// TIA Portal project "Proyecto1" (V15)

(* hardware
DEVICE "S7-1200 station_1"  S7-1200 Station
   slot 0: "Rack_0"  S7-1200 Rack  Rack  V1.0
   slot 1: "PLC_1"  CPU 1214C AC/DC/Rly  6ES7 214-1BG40-0XB0  V4.2
   slot 3: "CB 1241 (RS485)"  CB 1241 (RS485)  6ES7 241-1CH30-1XB0  V1.0
DEVICE "HMI_1"  KTP600 Basic color PN
   slot 0: "HMI_1"  KTP600 Basic color PN  6AV6 647-0AD11-3AX0  12.0.0.0
   slot 1: "HMI_RT_1"  KTP600 Basic color PN  6AV6 647-0AD11-3AX0  12.0.0.0
   slot 5: "HMI_1.IE_CP_1"  PROFINET Interface  12.0.0.0
      slot 1: "Interfaz PROFINET_1"  PROFINET Interface
         slot 1: "Port_1"  Port
*)

// ===== PLC "PLC_1"  CPU 1214C AC/DC/Rly =====

VAR_GLOBAL   // PLC tag table "Tabla de variables estándar"
   "First Scan" AT %M1.0 : Bool;
   "Tag_1" AT %I0.1 : Bool;
   "Tag_2" AT %I0.2 : Bool;
   "Tag_3" AT %Q0.0 : Bool;
   "0.5 Hz clock" AT %M0.7 : Bool;
   "mHora" AT %M0.3 : Bool;
   "reset_hora_contador" AT %MW100 : Int;
END_VAR

TYPE "FLOW_PARA_DB"
   STRUCT
      "Process Values" : Struct
         Massflow : Real;
         Volumeflow : Real;
         Density : Real;
         Temperature : Real;
         "Frame temperature" : Real;
      END_STRUCT;
      "Identification data" : Struct
         "Sensor serial number" : String[20];
      END_STRUCT;
      Totalizer : Struct
         "Totalizer value" : Real;
         "Reset totalizer" : UInt := 1;
      END_STRUCT;
      "Device diagnostic" : Struct
         "Driver current" : Real;
         "Pick-up amplitude 1" : Real;
         "Pick-up amplitude 2" : Real;
         "Sensor frequency" : Real;
      END_STRUCT;
      "Zero Point adjustment" : Struct
         "Zero point duration" : UInt := 30;
         "Standard deviation" : Real;
         "Zero point offset value" : Real;
         "Zero point adjust progress" : UInt;
         "Zero point adjust status" : UInt;
         "Start Zero point adjustment" : UInt := 2;
      END_STRUCT;
      Setup : Struct
         "Flow direction" : UInt := 0;
         "Process noise damping" : UInt;
         "Low Massflow cutofff" : Real;
         "Low volumeflow cutoff" : Real;
      END_STRUCT;
      "Aerated Flow" : Struct
         "Aerated flow alarm limit" : UInt;
         "Aerated flow warning limit" : UInt;
         "Measurement sample time" : UInt;
         "Aerated flow filter" : UInt;
         "Filter time constant" : UInt;
         "Filter start hysteresis" : Real;
         "Minimum filtering time" : UInt;
      END_STRUCT;
      Alarms : Struct
         "Alarm group 1" : UDInt;
         "Alarm group 2" : UDInt;
      END_STRUCT;
      "Access level" : Struct
         "Access level" : UInt;
         "Access Password" : UInt := 2457;
      END_STRUCT;
      HMI_Commands : Struct
         CMD_200 : Bool;
         CMD_210 : Bool;
         CMD_220 : Bool;
         CMD_230 : Bool;
         CMD_240 : Bool;
         CMD_250 : Bool;
         CMD_260 : Bool;
         CMD_280 : Bool;
         CMD_290 : Bool;
         CMD_420 : Bool;
         CMD_440 : Bool;
         CMD_450 : Bool;
         CMD_460 : Bool;
         CMD_490_log_in : Bool;
         CMD_491_log_out : Bool;
      END_STRUCT;
      FB_Interface : Struct
         Input : Struct
            MB_ADDR : UInt := 3;
            CMD_IN : Int;
         END_STRUCT;
         Output : Struct
            CMD_INPR : Bool;
            CMD_ERR : Bool;
            ERR_MB_MASTER : Bool;
            STATUS_MB_MASTER : Word;
         END_STRUCT;
         InOut : Struct
            CMD_EN : Bool;
         END_STRUCT;
      END_STRUCT;
   END_STRUCT;
END_TYPE

DATA_BLOCK "FECHA_Y_HORA"   // DB2
{ S7_Optimized_Access := 'TRUE' }
VERSION : 0.1
   VAR
      Local : DTL;
   END_VAR
BEGIN
END_DATA_BLOCK

DATA_BLOCK "CONTADOR_DB"   // DB3
{ S7_Optimized_Access := 'TRUE' }
VERSION : 0.1
// stored: InstanceOfName CONTADOR
"CONTADOR"
BEGIN
END_DATA_BLOCK

DATA_BLOCK "CONTADOR_NODE"   // DB5
{ S7_Optimized_Access := 'FALSE' }
VERSION : 0.1
   VAR
      cSecadero : Int;
      cHorno : Int;
   END_VAR
BEGIN
END_DATA_BLOCK

DATA_BLOCK "DB_FLOW_PARA"   // DB17
{ S7_Optimized_Access := 'FALSE' }
VERSION : 0.1
BEGIN
END_DATA_BLOCK

DATA_BLOCK "FC410_FC_MODBUS_DB"   // DB95
{ S7_Optimized_Access := 'TRUE' }
VERSION : 0.1
// stored: InstanceOfName FC410_MODBUS
"FC410_MODBUS"
BEGIN
END_DATA_BLOCK

// folder: System blocks/Program resources

DATA_BLOCK "CONTADOR_PIEZAS_SECADERO"   // DB1
{ S7_Optimized_Access := 'TRUE' }
AUTHOR : Simatic
FAMILY : IEC
NAME : CNTR
VERSION : 1.0
// stored: InstanceOfName IEC_COUNTER
"IEC_COUNTER"
BEGIN
END_DATA_BLOCK

DATA_BLOCK "CONTADOR_PIEZAS_HORNO"   // DB4
{ S7_Optimized_Access := 'TRUE' }
AUTHOR : Simatic
FAMILY : IEC
NAME : CNTR
VERSION : 1.0
// stored: InstanceOfName IEC_COUNTER
"IEC_COUNTER"
BEGIN
END_DATA_BLOCK

// folder: (top level)

FUNCTION_BLOCK "FC410_MODBUS"   // FB1, LAD
{ S7_Optimized_Access := 'TRUE' }
VERSION : 0.1
   VAR_INPUT
      CMD_IN : Int;
      MB_ADDR : UInt;
   END_VAR
   VAR_OUTPUT
      CMD_INPR : Bool;
      CMD_ERR : Bool;
      ERR_MB_MASTER : Bool;
      STATUS_MB_MASTER : Word;
   END_VAR
   VAR_IN_OUT
      CMD_EN : Bool;
      DB_PARA : "FLOW_PARA_DB";
   END_VAR
   VAR
      CMD_INPR_COUNT : USInt;
   END_VAR
   VAR_TEMP
      Temp_Length_Read : DInt;
      "Temp_String Help" : String[2];
      "Alarm Group 2_temp" : UDInt;
   END_VAR
   VAR_TEMP   // added for the SCL form of the ladder/FBD networks
      _w1 : Bool;
      _w2 : Bool;
   END_VAR
BEGIN

REGION Network 1: Command 200 - Read Process Values 1/3
   // Reading Massflow, Volumeflow and density
   // 
   // DATA_ADDR: Modbus adr.: 3000 + 3002 + 3004
   // DATA_LEN: 6 words
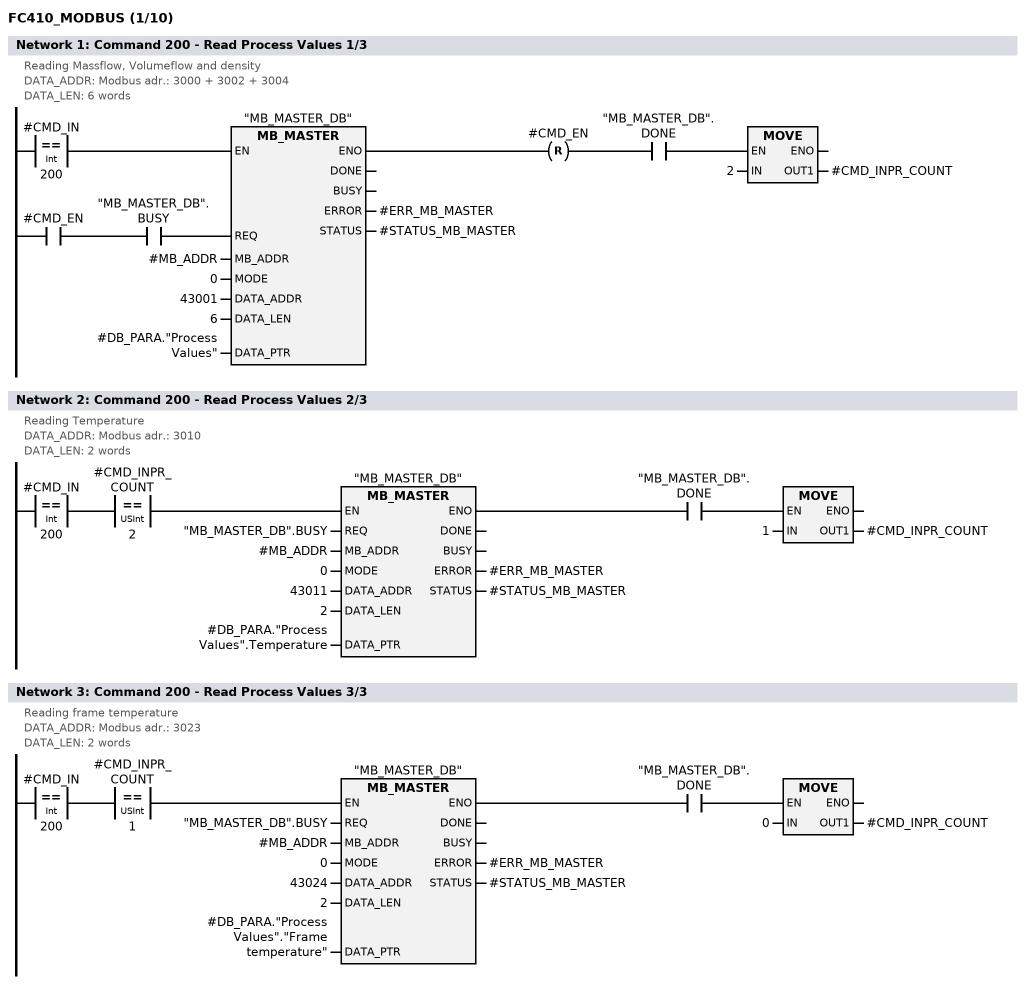
   // ENO of a box is taken as its EN; it also drops when the box reports an error
   #_w1 := #CMD_IN = 200;
   IF #_w1 THEN
       "MB_MASTER_DB"(REQ := #CMD_EN AND "MB_MASTER_DB".BUSY,   // MB_MASTER
                      MB_ADDR := #MB_ADDR,
                      MODE := 0,
                      DATA_ADDR := 43001,
                      DATA_LEN := 6,
                      DATA_PTR := #DB_PARA."Process Values",
                      ERROR => #ERR_MB_MASTER,
                      STATUS => #STATUS_MB_MASTER);
       #CMD_EN := FALSE;
   END_IF;
   IF #_w1 AND "MB_MASTER_DB".DONE THEN #CMD_INPR_COUNT := 2; END_IF;
END_REGION

REGION Network 2: Command 200 - Read Process Values 2/3
   // Reading Temperature
   // 
   // DATA_ADDR: Modbus adr.: 3010
   // DATA_LEN: 2 words
   // ENO of a box is taken as its EN; it also drops when the box reports an error
   #_w1 := (#CMD_IN = 200) AND (#CMD_INPR_COUNT = 2);
   IF #_w1 THEN
       "MB_MASTER_DB"(REQ := "MB_MASTER_DB".BUSY,   // MB_MASTER
                      MB_ADDR := #MB_ADDR,
                      MODE := 0,
                      DATA_ADDR := 43011,
                      DATA_LEN := 2,
                      DATA_PTR := #DB_PARA."Process Values".Temperature,
                      ERROR => #ERR_MB_MASTER,
                      STATUS => #STATUS_MB_MASTER);
   END_IF;
   IF #_w1 AND "MB_MASTER_DB".DONE THEN #CMD_INPR_COUNT := 1; END_IF;
END_REGION

REGION Network 3: Command 200 - Read Process Values 3/3
   // Reading frame temperature
   // 
   // DATA_ADDR: Modbus adr.: 3023
   // DATA_LEN: 2 words
   // ENO of a box is taken as its EN; it also drops when the box reports an error
   #_w1 := (#CMD_IN = 200) AND (#CMD_INPR_COUNT = 1);
   IF #_w1 THEN
       "MB_MASTER_DB"(REQ := "MB_MASTER_DB".BUSY,   // MB_MASTER
                      MB_ADDR := #MB_ADDR,
                      MODE := 0,
                      DATA_ADDR := 43024,
                      DATA_LEN := 2,
                      DATA_PTR := #DB_PARA."Process Values"."Frame temperature",
                      ERROR => #ERR_MB_MASTER,
                      STATUS => #STATUS_MB_MASTER);
   END_IF;
   IF #_w1 AND "MB_MASTER_DB".DONE THEN #CMD_INPR_COUNT := 0; END_IF;
END_REGION

REGION Network 4: Command 210 - Read Sensor Serial Number
   // DATA_ADDR: Modbus adr.: 4033
   // DATA_LEN: 10 words
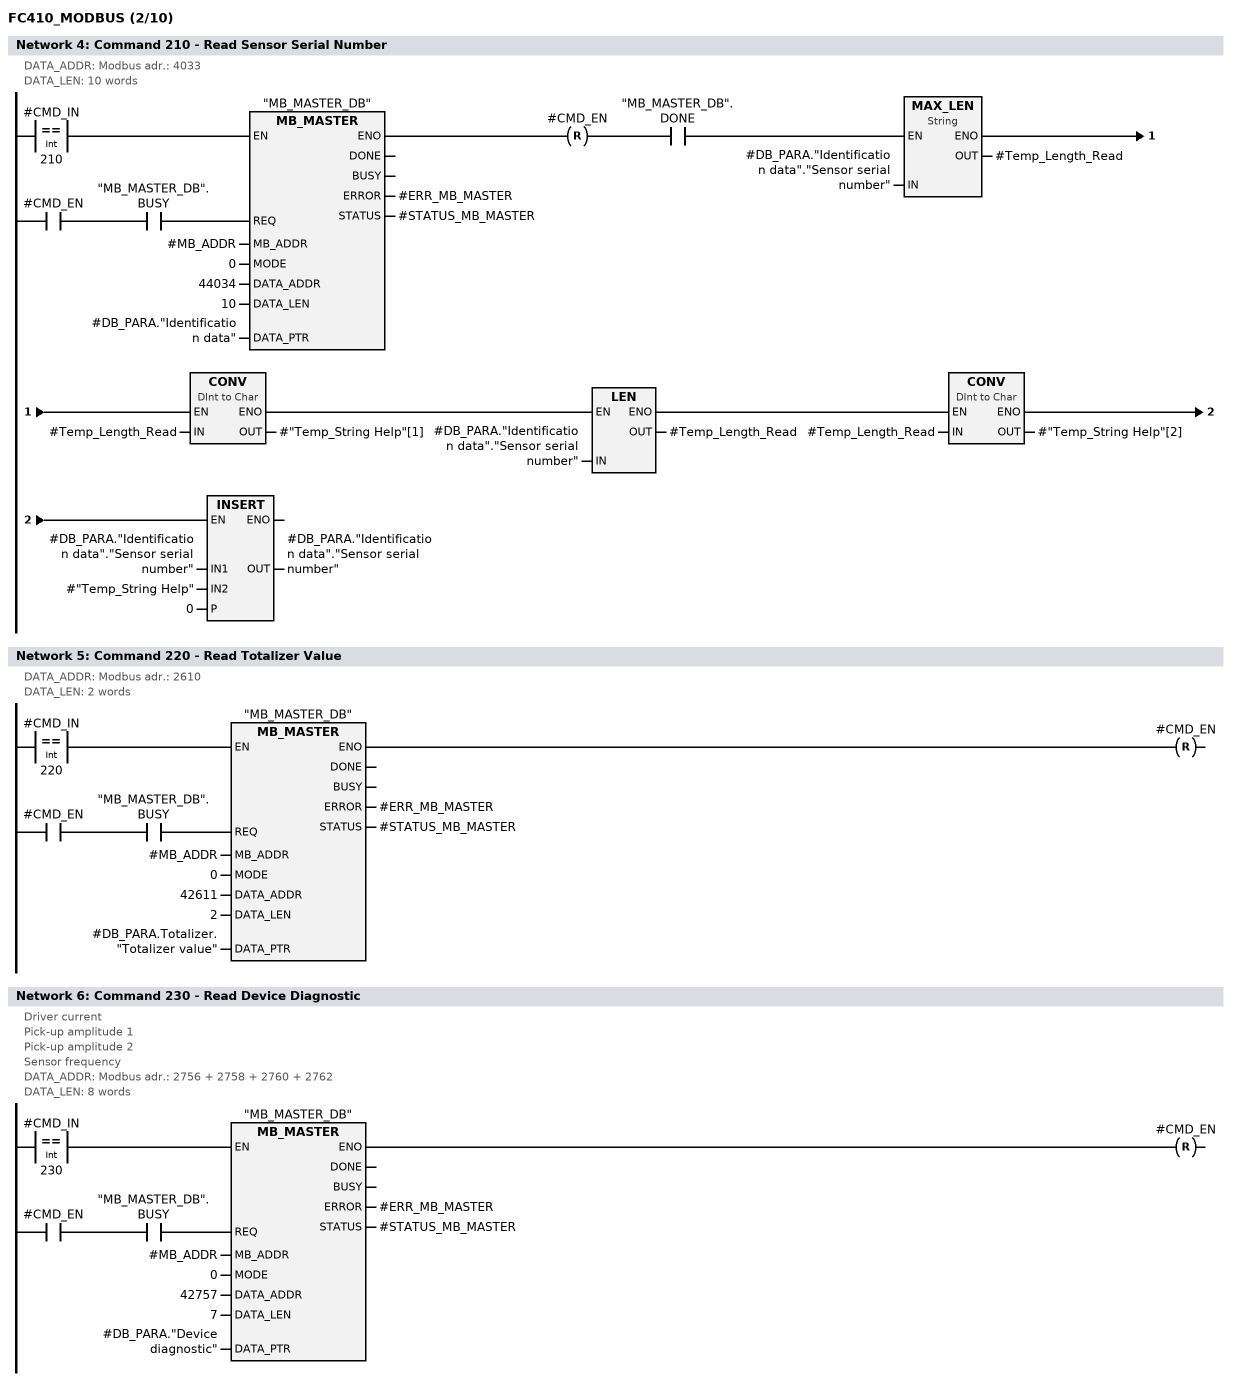
   // ENO of a box is taken as its EN; it also drops when the box reports an error
   #_w1 := #CMD_IN = 210;
   IF #_w1 THEN
       "MB_MASTER_DB"(REQ := #CMD_EN AND "MB_MASTER_DB".BUSY,   // MB_MASTER
                      MB_ADDR := #MB_ADDR,
                      MODE := 0,
                      DATA_ADDR := 44034,
                      DATA_LEN := 10,
                      DATA_PTR := #DB_PARA."Identification data",
                      ERROR => #ERR_MB_MASTER,
                      STATUS => #STATUS_MB_MASTER);
       #CMD_EN := FALSE;
   END_IF;
   #_w2 := #_w1 AND "MB_MASTER_DB".DONE;
   IF #_w2 THEN
       MAX_LEN(in := #DB_PARA."Identification data"."Sensor serial number", out => #Temp_Length_Read);
       #"Temp_String Help"[1] := DINT_TO_CHAR(#Temp_Length_Read);
       #Temp_Length_Read := LEN(IN := #DB_PARA."Identification data"."Sensor serial number");
       #"Temp_String Help"[2] := DINT_TO_CHAR(#Temp_Length_Read);
       #DB_PARA."Identification data"."Sensor serial number" := INSERT(IN1 := #DB_PARA."Identification data"."Sensor serial number",
                               IN2 := #"Temp_String Help",
                               P := 0);
   END_IF;
END_REGION

REGION Network 5: Command 220 - Read Totalizer Value
   // DATA_ADDR: Modbus adr.: 2610
   // DATA_LEN: 2 words
   // ENO of a box is taken as its EN; it also drops when the box reports an error
   IF #CMD_IN = 220 THEN
       "MB_MASTER_DB"(REQ := #CMD_EN AND "MB_MASTER_DB".BUSY,   // MB_MASTER
                      MB_ADDR := #MB_ADDR,
                      MODE := 0,
                      DATA_ADDR := 42611,
                      DATA_LEN := 2,
                      DATA_PTR := #DB_PARA.Totalizer."Totalizer value",
                      ERROR => #ERR_MB_MASTER,
                      STATUS => #STATUS_MB_MASTER);
       #CMD_EN := FALSE;
   END_IF;
END_REGION

REGION Network 6: Command 230 - Read Device Diagnostic
   // Driver current
   // Pick-up amplitude 1
   // Pick-up amplitude 2
   // Sensor frequency
   // 
   // 
   // DATA_ADDR: Modbus adr.: 2756 + 2758 + 2760 + 2762
   // DATA_LEN: 8 words
   // ENO of a box is taken as its EN; it also drops when the box reports an error
   IF #CMD_IN = 230 THEN
       "MB_MASTER_DB"(REQ := #CMD_EN AND "MB_MASTER_DB".BUSY,   // MB_MASTER
                      MB_ADDR := #MB_ADDR,
                      MODE := 0,
                      DATA_ADDR := 42757,
                      DATA_LEN := 7,
                      DATA_PTR := #DB_PARA."Device diagnostic",
                      ERROR => #ERR_MB_MASTER,
                      STATUS => #STATUS_MB_MASTER);
       #CMD_EN := FALSE;
   END_IF;
END_REGION

REGION Network 7: Command 240 - Read Zero Point Values 1/3
   // Read Zero point duration
   // 
   // DATA_ADDR: Modbus adr.: 2135
   // DATA_LEN: 1 words
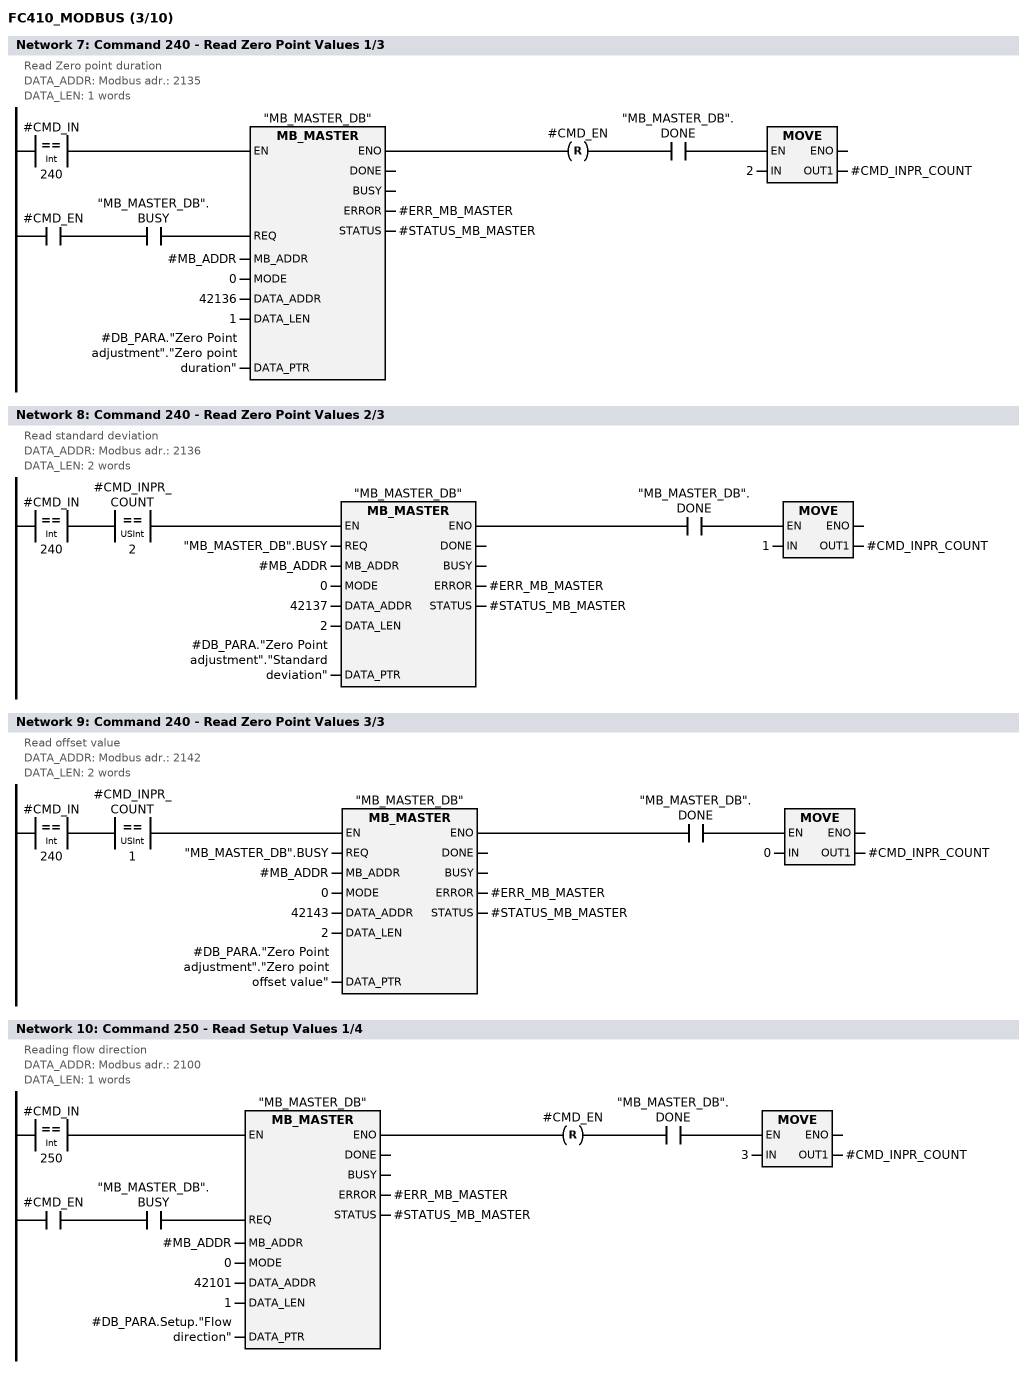
   // ENO of a box is taken as its EN; it also drops when the box reports an error
   #_w1 := #CMD_IN = 240;
   IF #_w1 THEN
       "MB_MASTER_DB"(REQ := #CMD_EN AND "MB_MASTER_DB".BUSY,   // MB_MASTER
                      MB_ADDR := #MB_ADDR,
                      MODE := 0,
                      DATA_ADDR := 42136,
                      DATA_LEN := 1,
                      DATA_PTR := #DB_PARA."Zero Point adjustment"."Zero point duration",
                      ERROR => #ERR_MB_MASTER,
                      STATUS => #STATUS_MB_MASTER);
       #CMD_EN := FALSE;
   END_IF;
   IF #_w1 AND "MB_MASTER_DB".DONE THEN #CMD_INPR_COUNT := 2; END_IF;
END_REGION

REGION Network 8: Command 240 - Read Zero Point Values 2/3
   // Read standard deviation
   // 
   // DATA_ADDR: Modbus adr.: 2136
   // DATA_LEN: 2 words
   // ENO of a box is taken as its EN; it also drops when the box reports an error
   #_w1 := (#CMD_IN = 240) AND (#CMD_INPR_COUNT = 2);
   IF #_w1 THEN
       "MB_MASTER_DB"(REQ := "MB_MASTER_DB".BUSY,   // MB_MASTER
                      MB_ADDR := #MB_ADDR,
                      MODE := 0,
                      DATA_ADDR := 42137,
                      DATA_LEN := 2,
                      DATA_PTR := #DB_PARA."Zero Point adjustment"."Standard deviation",
                      ERROR => #ERR_MB_MASTER,
                      STATUS => #STATUS_MB_MASTER);
   END_IF;
   IF #_w1 AND "MB_MASTER_DB".DONE THEN #CMD_INPR_COUNT := 1; END_IF;
END_REGION

REGION Network 9: Command 240 - Read Zero Point Values 3/3
   // Read offset value
   // 
   // DATA_ADDR: Modbus adr.: 2142
   // DATA_LEN: 2 words
   // ENO of a box is taken as its EN; it also drops when the box reports an error
   #_w1 := (#CMD_IN = 240) AND (#CMD_INPR_COUNT = 1);
   IF #_w1 THEN
       "MB_MASTER_DB"(REQ := "MB_MASTER_DB".BUSY,   // MB_MASTER
                      MB_ADDR := #MB_ADDR,
                      MODE := 0,
                      DATA_ADDR := 42143,
                      DATA_LEN := 2,
                      DATA_PTR := #DB_PARA."Zero Point adjustment"."Zero point offset value",
                      ERROR => #ERR_MB_MASTER,
                      STATUS => #STATUS_MB_MASTER);
   END_IF;
   IF #_w1 AND "MB_MASTER_DB".DONE THEN #CMD_INPR_COUNT := 0; END_IF;
END_REGION

REGION Network 10: Command 250 - Read Setup Values 1/4
   // Reading flow direction
   // 
   // DATA_ADDR: Modbus adr.: 2100
   // DATA_LEN: 1 words
   // ENO of a box is taken as its EN; it also drops when the box reports an error
   #_w1 := #CMD_IN = 250;
   IF #_w1 THEN
       "MB_MASTER_DB"(REQ := #CMD_EN AND "MB_MASTER_DB".BUSY,   // MB_MASTER
                      MB_ADDR := #MB_ADDR,
                      MODE := 0,
                      DATA_ADDR := 42101,
                      DATA_LEN := 1,
                      DATA_PTR := #DB_PARA.Setup."Flow direction",
                      ERROR => #ERR_MB_MASTER,
                      STATUS => #STATUS_MB_MASTER);
       #CMD_EN := FALSE;
   END_IF;
   IF #_w1 AND "MB_MASTER_DB".DONE THEN #CMD_INPR_COUNT := 3; END_IF;
END_REGION

REGION Network 11: Command 250 - Read Setup Values 2/4
   // Reading process noise damping
   // 
   // DATA_ADDR: Modbus adr.: 2130
   // DATA_LEN: 1 words
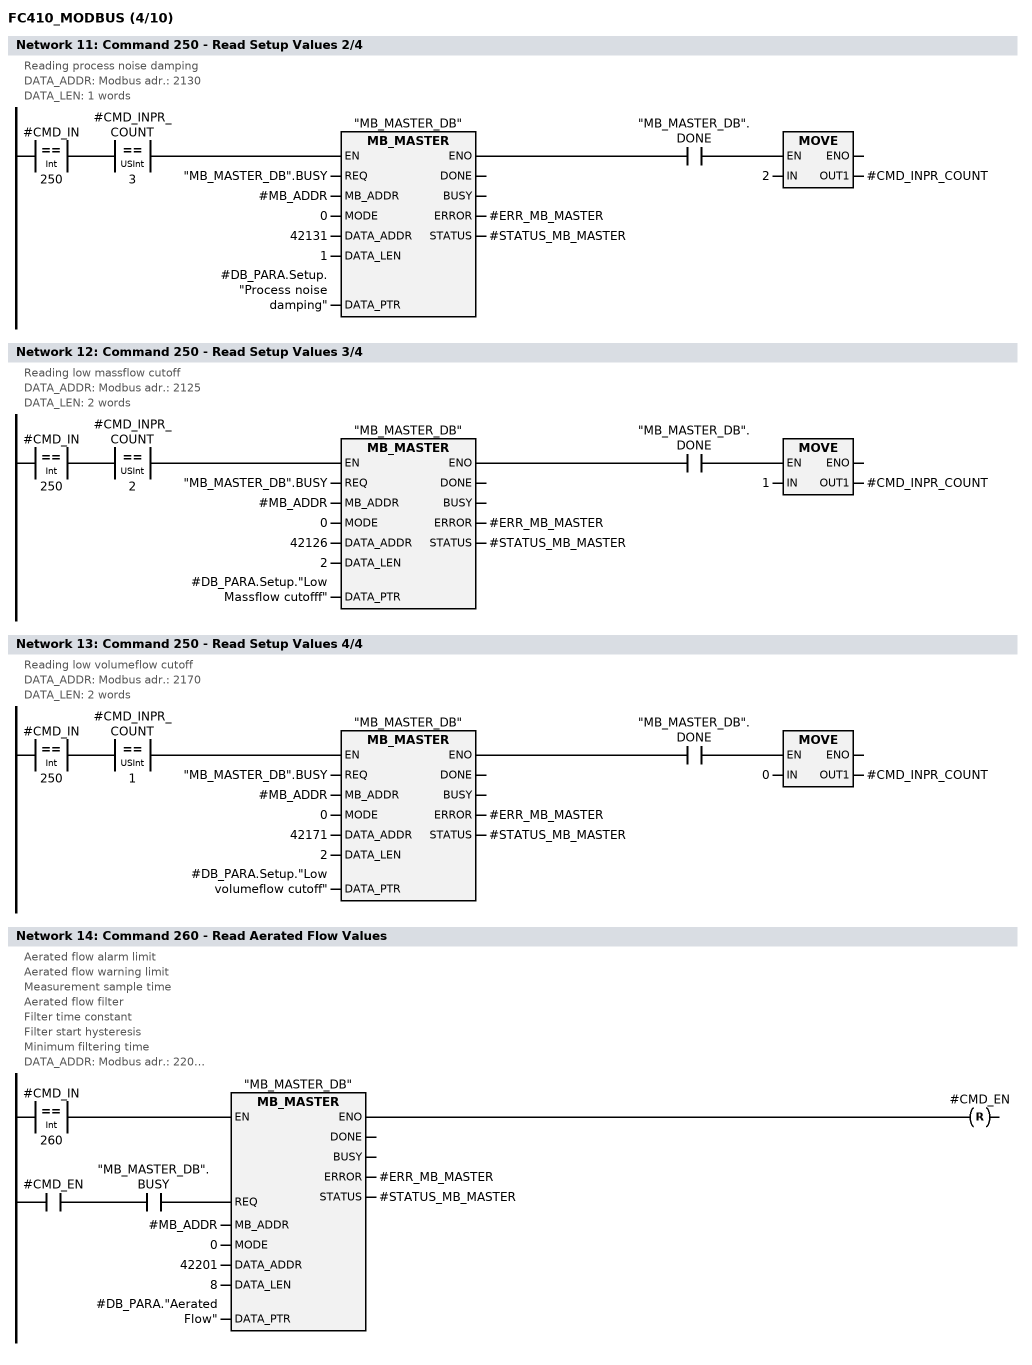
   // ENO of a box is taken as its EN; it also drops when the box reports an error
   #_w1 := (#CMD_IN = 250) AND (#CMD_INPR_COUNT = 3);
   IF #_w1 THEN
       "MB_MASTER_DB"(REQ := "MB_MASTER_DB".BUSY,   // MB_MASTER
                      MB_ADDR := #MB_ADDR,
                      MODE := 0,
                      DATA_ADDR := 42131,
                      DATA_LEN := 1,
                      DATA_PTR := #DB_PARA.Setup."Process noise damping",
                      ERROR => #ERR_MB_MASTER,
                      STATUS => #STATUS_MB_MASTER);
   END_IF;
   IF #_w1 AND "MB_MASTER_DB".DONE THEN #CMD_INPR_COUNT := 2; END_IF;
END_REGION

REGION Network 12: Command 250 - Read Setup Values 3/4
   // Reading low massflow cutoff
   // 
   // DATA_ADDR: Modbus adr.: 2125
   // DATA_LEN: 2 words
   // ENO of a box is taken as its EN; it also drops when the box reports an error
   #_w1 := (#CMD_IN = 250) AND (#CMD_INPR_COUNT = 2);
   IF #_w1 THEN
       "MB_MASTER_DB"(REQ := "MB_MASTER_DB".BUSY,   // MB_MASTER
                      MB_ADDR := #MB_ADDR,
                      MODE := 0,
                      DATA_ADDR := 42126,
                      DATA_LEN := 2,
                      DATA_PTR := #DB_PARA.Setup."Low Massflow cutofff",
                      ERROR => #ERR_MB_MASTER,
                      STATUS => #STATUS_MB_MASTER);
   END_IF;
   IF #_w1 AND "MB_MASTER_DB".DONE THEN #CMD_INPR_COUNT := 1; END_IF;
END_REGION

REGION Network 13: Command 250 - Read Setup Values 4/4
   // Reading low volumeflow cutoff
   // 
   // DATA_ADDR: Modbus adr.: 2170
   // DATA_LEN: 2 words
   // ENO of a box is taken as its EN; it also drops when the box reports an error
   #_w1 := (#CMD_IN = 250) AND (#CMD_INPR_COUNT = 1);
   IF #_w1 THEN
       "MB_MASTER_DB"(REQ := "MB_MASTER_DB".BUSY,   // MB_MASTER
                      MB_ADDR := #MB_ADDR,
                      MODE := 0,
                      DATA_ADDR := 42171,
                      DATA_LEN := 2,
                      DATA_PTR := #DB_PARA.Setup."Low volumeflow cutoff",
                      ERROR => #ERR_MB_MASTER,
                      STATUS => #STATUS_MB_MASTER);
   END_IF;
   IF #_w1 AND "MB_MASTER_DB".DONE THEN #CMD_INPR_COUNT := 0; END_IF;
END_REGION

REGION Network 14: Command 260 - Read Aerated Flow Values
   // Aerated flow alarm limit
   // Aerated flow warning limit
   // Measurement sample time
   // Aerated flow filter
   // Filter time constant
   // Filter start hysteresis
   // Minimum filtering time
   // 
   // DATA_ADDR: Modbus adr.: 2200
   // DATA_LEN: 8 words
   // ENO of a box is taken as its EN; it also drops when the box reports an error
   IF #CMD_IN = 260 THEN
       "MB_MASTER_DB"(REQ := #CMD_EN AND "MB_MASTER_DB".BUSY,   // MB_MASTER
                      MB_ADDR := #MB_ADDR,
                      MODE := 0,
                      DATA_ADDR := 42201,
                      DATA_LEN := 8,
                      DATA_PTR := #DB_PARA."Aerated Flow",
                      ERROR => #ERR_MB_MASTER,
                      STATUS => #STATUS_MB_MASTER);
       #CMD_EN := FALSE;
   END_IF;
END_REGION

REGION Network 15: Command 280 - Read Alarm Status
   // Alarm group 1
   // Alarm group 2
   // 
   // DATA_ADDR: Modbus adr.: 3012
   // DATA_LEN: 4 words
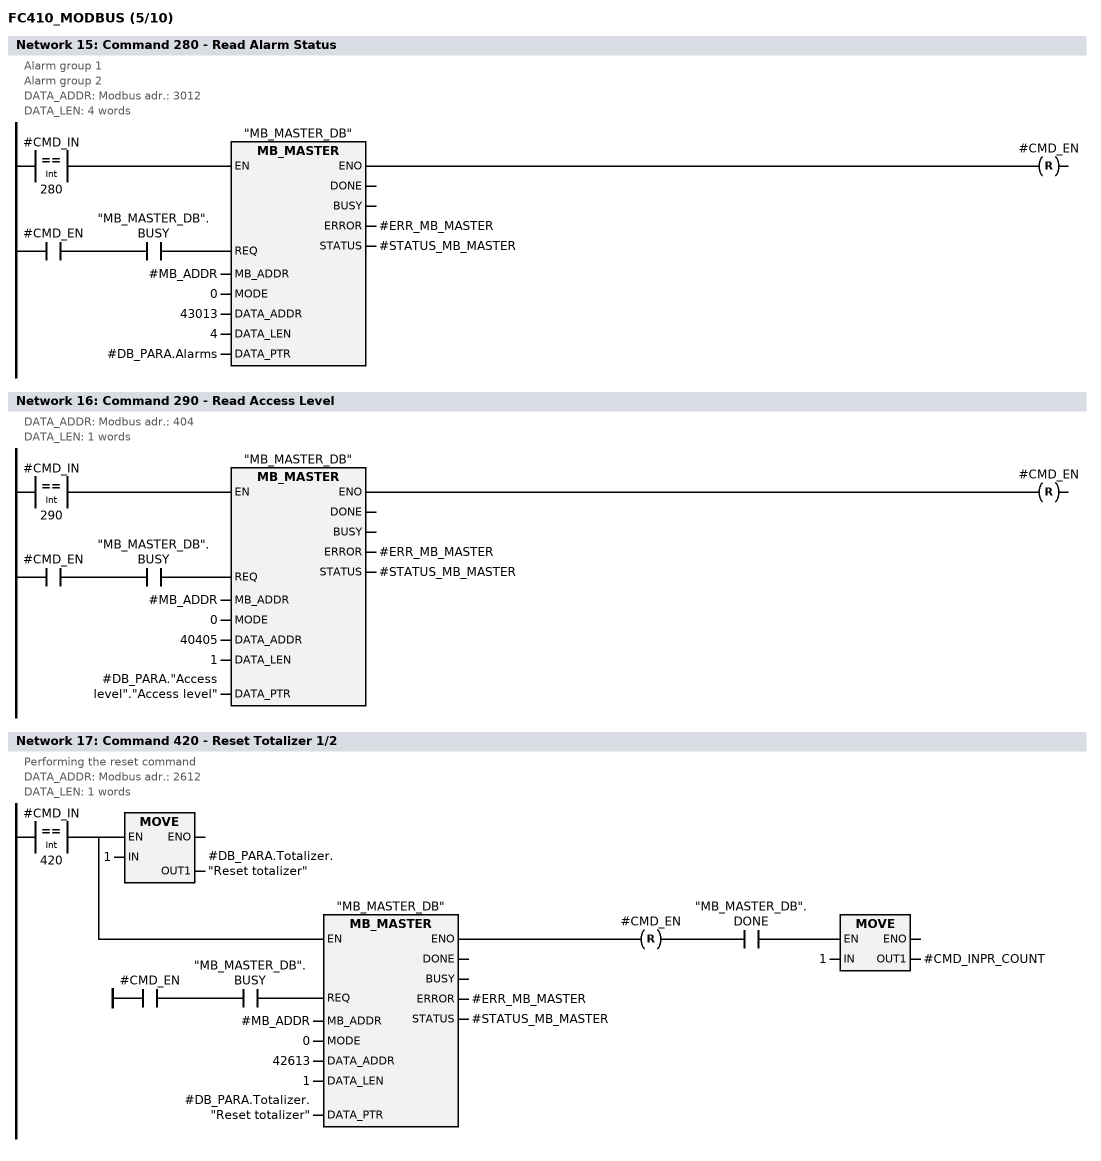
   // ENO of a box is taken as its EN; it also drops when the box reports an error
   IF #CMD_IN = 280 THEN
       "MB_MASTER_DB"(REQ := #CMD_EN AND "MB_MASTER_DB".BUSY,   // MB_MASTER
                      MB_ADDR := #MB_ADDR,
                      MODE := 0,
                      DATA_ADDR := 43013,
                      DATA_LEN := 4,
                      DATA_PTR := #DB_PARA.Alarms,
                      ERROR => #ERR_MB_MASTER,
                      STATUS => #STATUS_MB_MASTER);
       #CMD_EN := FALSE;
   END_IF;
END_REGION

REGION Network 16: Command 290 - Read Access Level
   // DATA_ADDR: Modbus adr.: 404
   // DATA_LEN: 1 words
   // ENO of a box is taken as its EN; it also drops when the box reports an error
   IF #CMD_IN = 290 THEN
       "MB_MASTER_DB"(REQ := #CMD_EN AND "MB_MASTER_DB".BUSY,   // MB_MASTER
                      MB_ADDR := #MB_ADDR,
                      MODE := 0,
                      DATA_ADDR := 40405,
                      DATA_LEN := 1,
                      DATA_PTR := #DB_PARA."Access level"."Access level",
                      ERROR => #ERR_MB_MASTER,
                      STATUS => #STATUS_MB_MASTER);
       #CMD_EN := FALSE;
   END_IF;
END_REGION

REGION Network 17: Command 420 - Reset Totalizer 1/2
   // Performing the reset command
   // 
   // DATA_ADDR: Modbus adr.: 2612
   // DATA_LEN: 1 words
   // ENO of a box is taken as its EN; it also drops when the box reports an error
   #_w1 := #CMD_IN = 420;
   IF #_w1 THEN
       #DB_PARA.Totalizer."Reset totalizer" := 1;
       "MB_MASTER_DB"(REQ := #CMD_EN AND "MB_MASTER_DB".BUSY,   // MB_MASTER
                      MB_ADDR := #MB_ADDR,
                      MODE := 0,
                      DATA_ADDR := 42613,
                      DATA_LEN := 1,
                      DATA_PTR := #DB_PARA.Totalizer."Reset totalizer",
                      ERROR => #ERR_MB_MASTER,
                      STATUS => #STATUS_MB_MASTER);
       #CMD_EN := FALSE;
   END_IF;
   IF #_w1 AND "MB_MASTER_DB".DONE THEN #CMD_INPR_COUNT := 1; END_IF;
END_REGION

REGION Network 18: Command 420 - Reset Totalizer 2/2
   // Reading the totalizer to verify reset
   // 
   // DATA_ADDR: Modbus adr.: 2610
   // DATA_LEN: 2 words
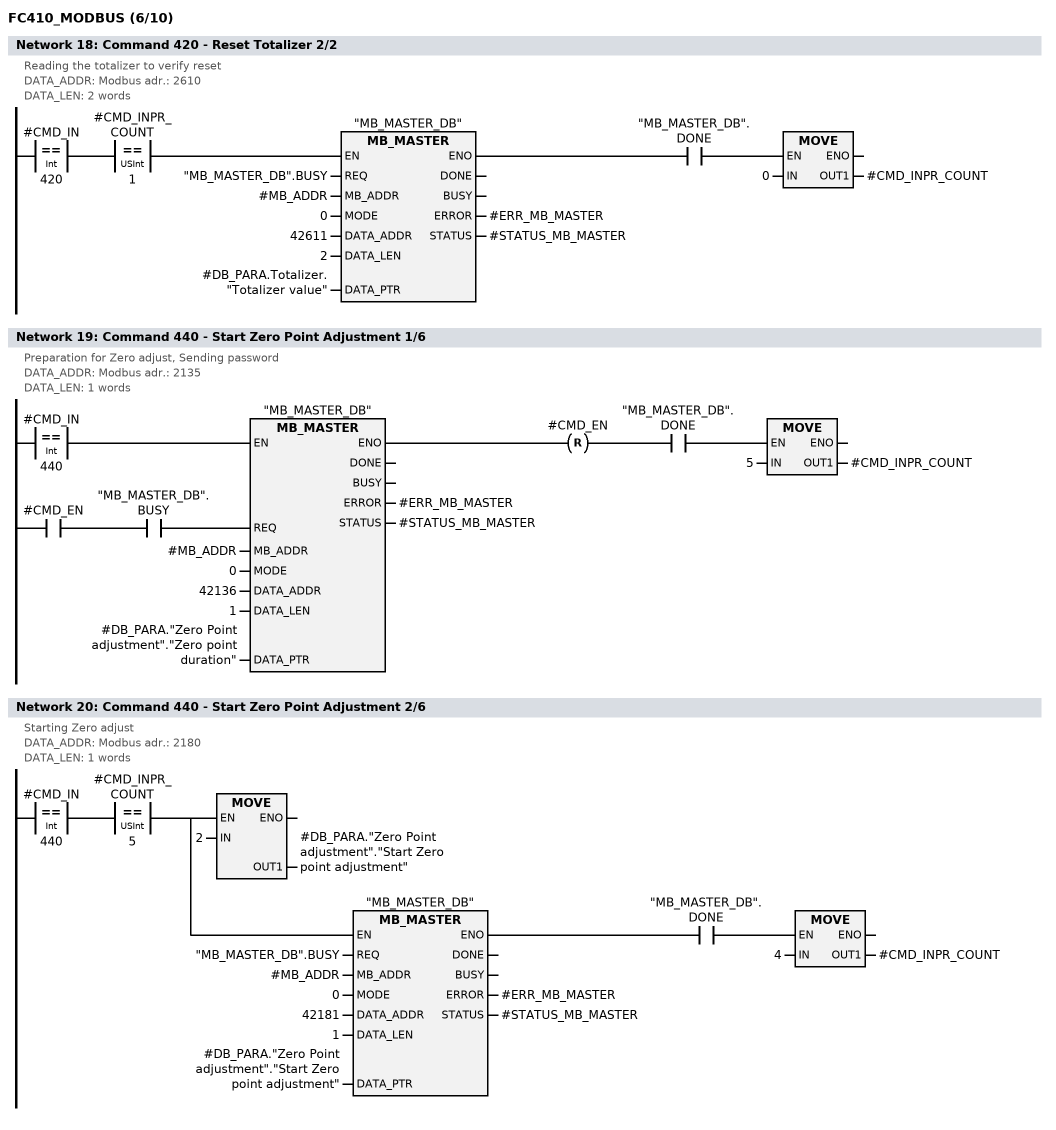
   // ENO of a box is taken as its EN; it also drops when the box reports an error
   #_w1 := (#CMD_IN = 420) AND (#CMD_INPR_COUNT = 1);
   IF #_w1 THEN
       "MB_MASTER_DB"(REQ := "MB_MASTER_DB".BUSY,   // MB_MASTER
                      MB_ADDR := #MB_ADDR,
                      MODE := 0,
                      DATA_ADDR := 42611,
                      DATA_LEN := 2,
                      DATA_PTR := #DB_PARA.Totalizer."Totalizer value",
                      ERROR => #ERR_MB_MASTER,
                      STATUS => #STATUS_MB_MASTER);
   END_IF;
   IF #_w1 AND "MB_MASTER_DB".DONE THEN #CMD_INPR_COUNT := 0; END_IF;
END_REGION

REGION Network 19: Command 440 - Start Zero Point Adjustment 1/6
   // Preparation for Zero adjust, Sending password
   // 
   // DATA_ADDR: Modbus adr.: 2135
   // DATA_LEN: 1 words
   // ENO of a box is taken as its EN; it also drops when the box reports an error
   #_w1 := #CMD_IN = 440;
   IF #_w1 THEN
       "MB_MASTER_DB"(REQ := #CMD_EN AND "MB_MASTER_DB".BUSY,   // MB_MASTER
                      MB_ADDR := #MB_ADDR,
                      MODE := 0,
                      DATA_ADDR := 42136,
                      DATA_LEN := 1,
                      DATA_PTR := #DB_PARA."Zero Point adjustment"."Zero point duration",
                      ERROR => #ERR_MB_MASTER,
                      STATUS => #STATUS_MB_MASTER);
       #CMD_EN := FALSE;
   END_IF;
   IF #_w1 AND "MB_MASTER_DB".DONE THEN #CMD_INPR_COUNT := 5; END_IF;
END_REGION

REGION Network 20: Command 440 - Start Zero Point Adjustment 2/6
   // Starting Zero adjust
   // 
   // DATA_ADDR: Modbus adr.: 2180
   // DATA_LEN: 1 words
   // ENO of a box is taken as its EN; it also drops when the box reports an error
   #_w1 := (#CMD_IN = 440) AND (#CMD_INPR_COUNT = 5);
   IF #_w1 THEN
       #DB_PARA."Zero Point adjustment"."Start Zero point adjustment" := 2;
       "MB_MASTER_DB"(REQ := "MB_MASTER_DB".BUSY,   // MB_MASTER
                      MB_ADDR := #MB_ADDR,
                      MODE := 0,
                      DATA_ADDR := 42181,
                      DATA_LEN := 1,
                      DATA_PTR := #DB_PARA."Zero Point adjustment"."Start Zero point adjustment",
                      ERROR => #ERR_MB_MASTER,
                      STATUS => #STATUS_MB_MASTER);
   END_IF;
   IF #_w1 AND "MB_MASTER_DB".DONE THEN #CMD_INPR_COUNT := 4; END_IF;
END_REGION

REGION Network 21: Command 440 - Start Zero Point Adjustment 3/6
   // Read ZeroAdj to ensure its started.
   // 
   // DATA_ADDR: Modbus adr.: 2180
   // DATA_LEN: 1 words
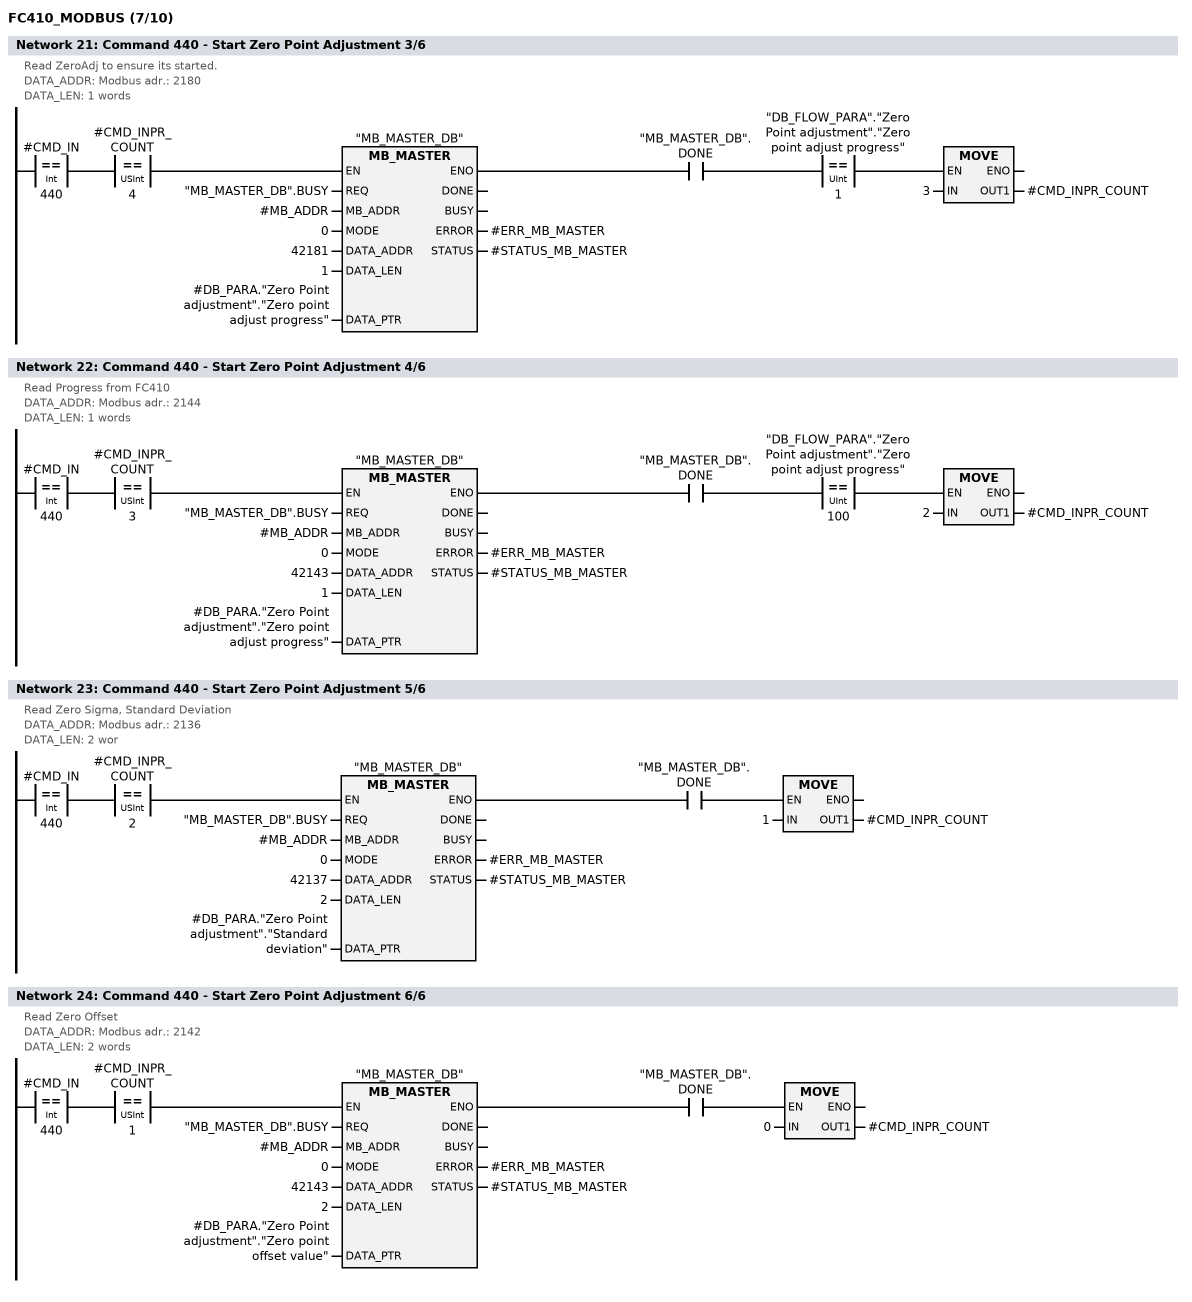
   // ENO of a box is taken as its EN; it also drops when the box reports an error
   #_w1 := (#CMD_IN = 440) AND (#CMD_INPR_COUNT = 4);
   IF #_w1 THEN
       "MB_MASTER_DB"(REQ := "MB_MASTER_DB".BUSY,   // MB_MASTER
                      MB_ADDR := #MB_ADDR,
                      MODE := 0,
                      DATA_ADDR := 42181,
                      DATA_LEN := 1,
                      DATA_PTR := #DB_PARA."Zero Point adjustment"."Zero point adjust progress",
                      ERROR => #ERR_MB_MASTER,
                      STATUS => #STATUS_MB_MASTER);
   END_IF;
   IF #_w1 AND "MB_MASTER_DB".DONE AND ("DB_FLOW_PARA"."Zero Point adjustment"."Zero point adjust progress" = 1) THEN
       #CMD_INPR_COUNT := 3;
   END_IF;
END_REGION

REGION Network 22: Command 440 - Start Zero Point Adjustment 4/6
   // Read Progress from FC410
   // 
   // DATA_ADDR: Modbus adr.: 2144
   // DATA_LEN: 1 words
   // ENO of a box is taken as its EN; it also drops when the box reports an error
   #_w1 := (#CMD_IN = 440) AND (#CMD_INPR_COUNT = 3);
   IF #_w1 THEN
       "MB_MASTER_DB"(REQ := "MB_MASTER_DB".BUSY,   // MB_MASTER
                      MB_ADDR := #MB_ADDR,
                      MODE := 0,
                      DATA_ADDR := 42143,
                      DATA_LEN := 1,
                      DATA_PTR := #DB_PARA."Zero Point adjustment"."Zero point adjust progress",
                      ERROR => #ERR_MB_MASTER,
                      STATUS => #STATUS_MB_MASTER);
   END_IF;
   IF #_w1 AND "MB_MASTER_DB".DONE AND ("DB_FLOW_PARA"."Zero Point adjustment"."Zero point adjust progress" = 100) THEN
       #CMD_INPR_COUNT := 2;
   END_IF;
END_REGION

REGION Network 23: Command 440 - Start Zero Point Adjustment 5/6
   // Read Zero Sigma, Standard Deviation
   // 
   // DATA_ADDR: Modbus adr.: 2136
   // DATA_LEN: 2 wor
   // ENO of a box is taken as its EN; it also drops when the box reports an error
   #_w1 := (#CMD_IN = 440) AND (#CMD_INPR_COUNT = 2);
   IF #_w1 THEN
       "MB_MASTER_DB"(REQ := "MB_MASTER_DB".BUSY,   // MB_MASTER
                      MB_ADDR := #MB_ADDR,
                      MODE := 0,
                      DATA_ADDR := 42137,
                      DATA_LEN := 2,
                      DATA_PTR := #DB_PARA."Zero Point adjustment"."Standard deviation",
                      ERROR => #ERR_MB_MASTER,
                      STATUS => #STATUS_MB_MASTER);
   END_IF;
   IF #_w1 AND "MB_MASTER_DB".DONE THEN #CMD_INPR_COUNT := 1; END_IF;
END_REGION

REGION Network 24: Command 440 - Start Zero Point Adjustment 6/6
   // Read Zero Offset
   // 
   // DATA_ADDR: Modbus adr.: 2142
   // DATA_LEN: 2 words
   // ENO of a box is taken as its EN; it also drops when the box reports an error
   #_w1 := (#CMD_IN = 440) AND (#CMD_INPR_COUNT = 1);
   IF #_w1 THEN
       "MB_MASTER_DB"(REQ := "MB_MASTER_DB".BUSY,   // MB_MASTER
                      MB_ADDR := #MB_ADDR,
                      MODE := 0,
                      DATA_ADDR := 42143,
                      DATA_LEN := 2,
                      DATA_PTR := #DB_PARA."Zero Point adjustment"."Zero point offset value",
                      ERROR => #ERR_MB_MASTER,
                      STATUS => #STATUS_MB_MASTER);
   END_IF;
   IF #_w1 AND "MB_MASTER_DB".DONE THEN #CMD_INPR_COUNT := 0; END_IF;
END_REGION

REGION Network 25: Command 450 - Write Setup Values 1/4
   // Writing flow direction
   // 
   // DATA_ADDR: Modbus adr.: 2100
   // DATA_LEN: 1 words
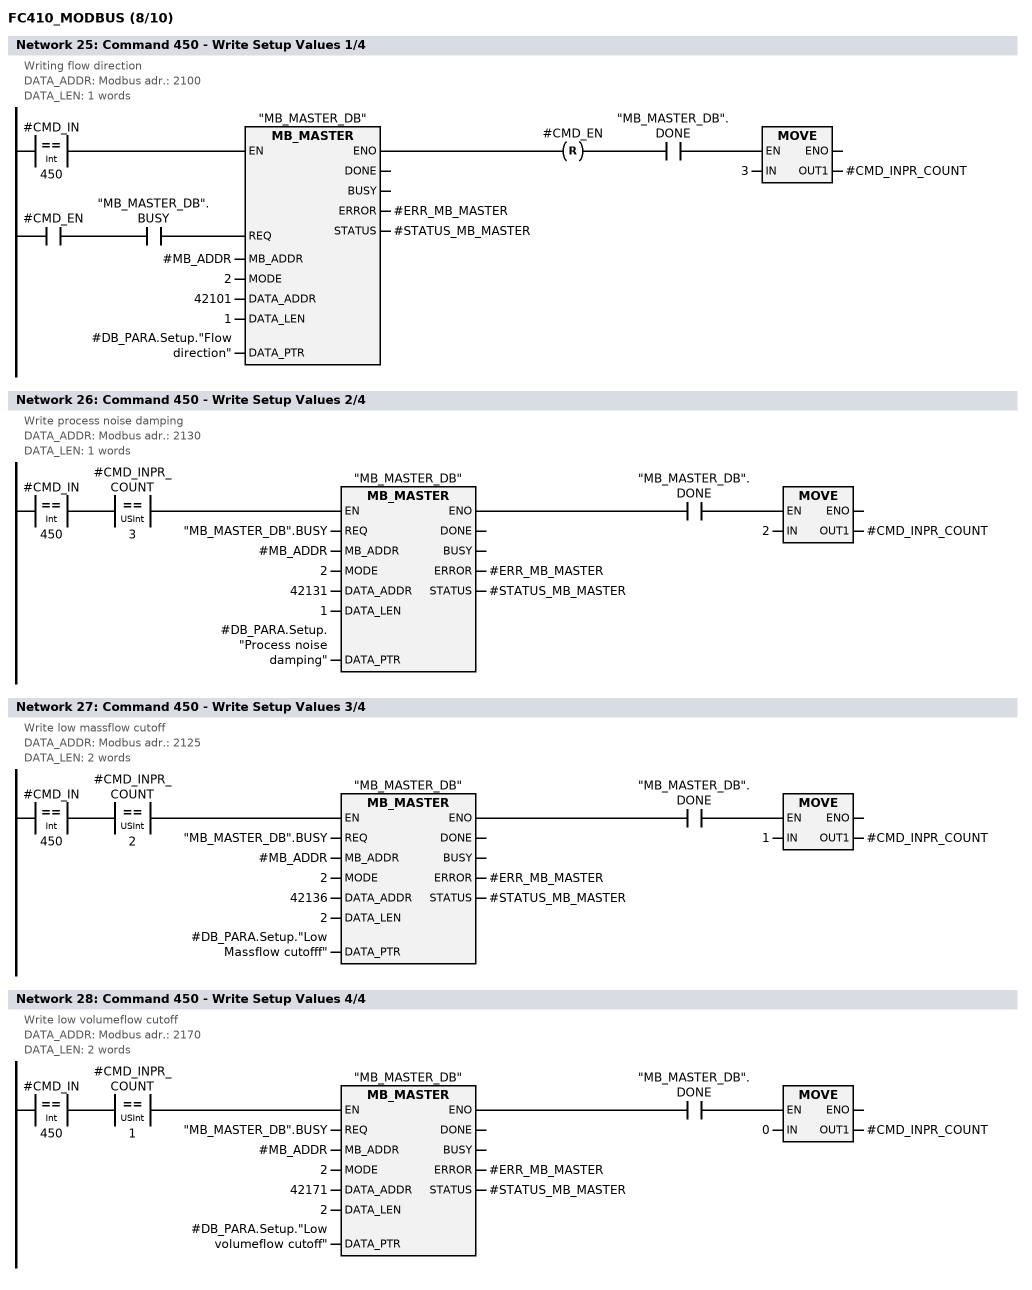
   // ENO of a box is taken as its EN; it also drops when the box reports an error
   #_w1 := #CMD_IN = 450;
   IF #_w1 THEN
       "MB_MASTER_DB"(REQ := #CMD_EN AND "MB_MASTER_DB".BUSY,   // MB_MASTER
                      MB_ADDR := #MB_ADDR,
                      MODE := 2,
                      DATA_ADDR := 42101,
                      DATA_LEN := 1,
                      DATA_PTR := #DB_PARA.Setup."Flow direction",
                      ERROR => #ERR_MB_MASTER,
                      STATUS => #STATUS_MB_MASTER);
       #CMD_EN := FALSE;
   END_IF;
   IF #_w1 AND "MB_MASTER_DB".DONE THEN #CMD_INPR_COUNT := 3; END_IF;
END_REGION

REGION Network 26: Command 450 - Write Setup Values 2/4
   // Write process noise damping
   // 
   // DATA_ADDR: Modbus adr.: 2130
   // DATA_LEN: 1 words
   // ENO of a box is taken as its EN; it also drops when the box reports an error
   #_w1 := (#CMD_IN = 450) AND (#CMD_INPR_COUNT = 3);
   IF #_w1 THEN
       "MB_MASTER_DB"(REQ := "MB_MASTER_DB".BUSY,   // MB_MASTER
                      MB_ADDR := #MB_ADDR,
                      MODE := 2,
                      DATA_ADDR := 42131,
                      DATA_LEN := 1,
                      DATA_PTR := #DB_PARA.Setup."Process noise damping",
                      ERROR => #ERR_MB_MASTER,
                      STATUS => #STATUS_MB_MASTER);
   END_IF;
   IF #_w1 AND "MB_MASTER_DB".DONE THEN #CMD_INPR_COUNT := 2; END_IF;
END_REGION

REGION Network 27: Command 450 - Write Setup Values 3/4
   // Write low massflow cutoff
   // 
   // DATA_ADDR: Modbus adr.: 2125
   // DATA_LEN: 2 words
   // ENO of a box is taken as its EN; it also drops when the box reports an error
   #_w1 := (#CMD_IN = 450) AND (#CMD_INPR_COUNT = 2);
   IF #_w1 THEN
       "MB_MASTER_DB"(REQ := "MB_MASTER_DB".BUSY,   // MB_MASTER
                      MB_ADDR := #MB_ADDR,
                      MODE := 2,
                      DATA_ADDR := 42136,
                      DATA_LEN := 2,
                      DATA_PTR := #DB_PARA.Setup."Low Massflow cutofff",
                      ERROR => #ERR_MB_MASTER,
                      STATUS => #STATUS_MB_MASTER);
   END_IF;
   IF #_w1 AND "MB_MASTER_DB".DONE THEN #CMD_INPR_COUNT := 1; END_IF;
END_REGION

REGION Network 28: Command 450 - Write Setup Values 4/4
   // Write low volumeflow cutoff
   // 
   // DATA_ADDR: Modbus adr.: 2170
   // DATA_LEN: 2 words
   // ENO of a box is taken as its EN; it also drops when the box reports an error
   #_w1 := (#CMD_IN = 450) AND (#CMD_INPR_COUNT = 1);
   IF #_w1 THEN
       "MB_MASTER_DB"(REQ := "MB_MASTER_DB".BUSY,   // MB_MASTER
                      MB_ADDR := #MB_ADDR,
                      MODE := 2,
                      DATA_ADDR := 42171,
                      DATA_LEN := 2,
                      DATA_PTR := #DB_PARA.Setup."Low volumeflow cutoff",
                      ERROR => #ERR_MB_MASTER,
                      STATUS => #STATUS_MB_MASTER);
   END_IF;
   IF #_w1 AND "MB_MASTER_DB".DONE THEN #CMD_INPR_COUNT := 0; END_IF;
END_REGION

REGION Network 29: Command 460 - Write Aerated Flow Values
   // DATA_ADDR: Modbus adr.: 2200 
   // DATA_LEN: 8 words
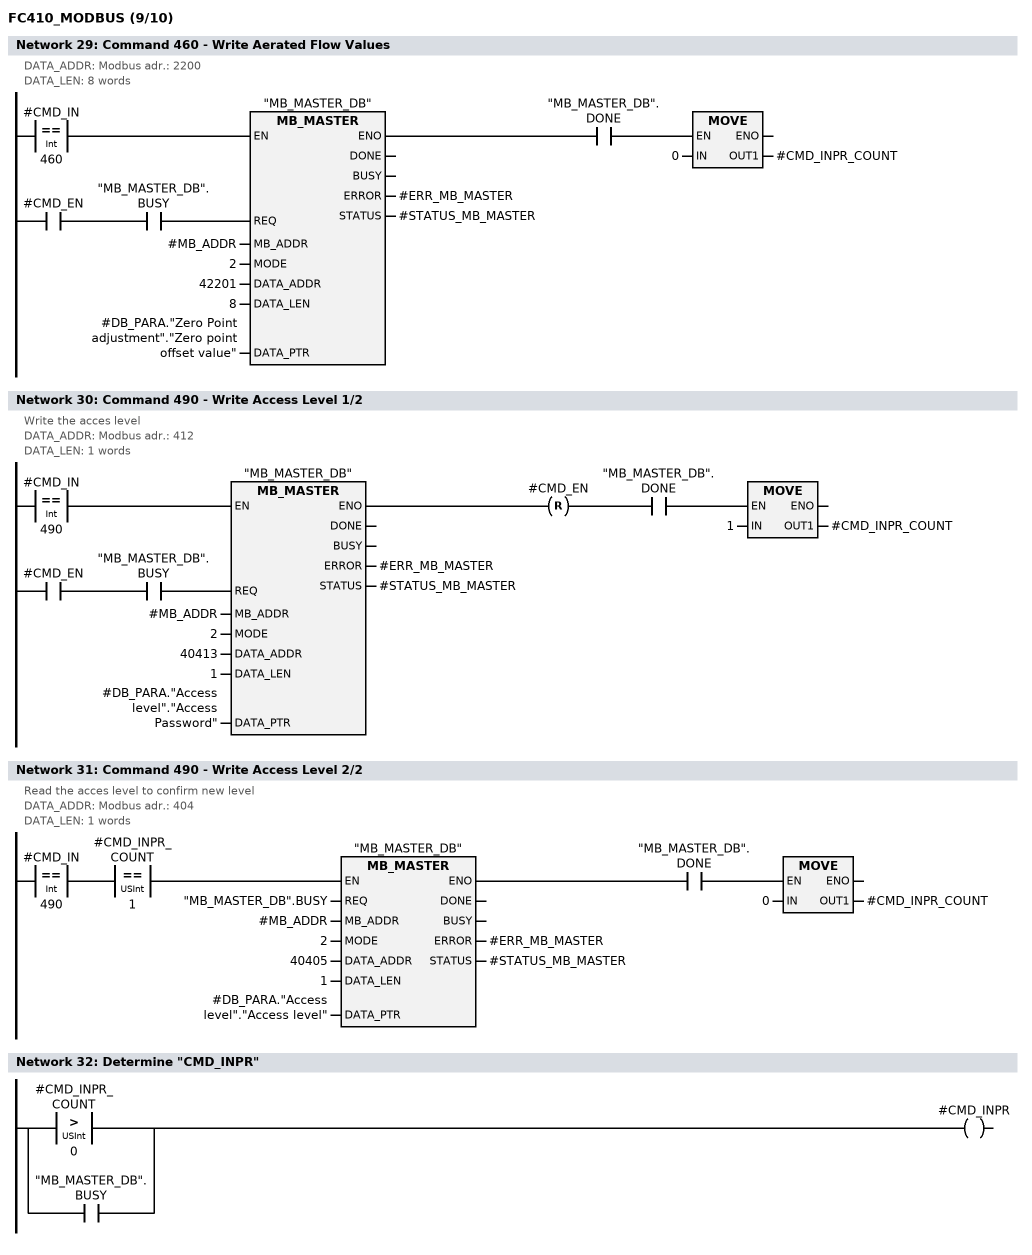
   // ENO of a box is taken as its EN; it also drops when the box reports an error
   #_w1 := #CMD_IN = 460;
   IF #_w1 THEN
       "MB_MASTER_DB"(REQ := #CMD_EN AND "MB_MASTER_DB".BUSY,   // MB_MASTER
                      MB_ADDR := #MB_ADDR,
                      MODE := 2,
                      DATA_ADDR := 42201,
                      DATA_LEN := 8,
                      DATA_PTR := #DB_PARA."Zero Point adjustment"."Zero point offset value",
                      ERROR => #ERR_MB_MASTER,
                      STATUS => #STATUS_MB_MASTER);
   END_IF;
   IF #_w1 AND "MB_MASTER_DB".DONE THEN #CMD_INPR_COUNT := 0; END_IF;
END_REGION

REGION Network 30: Command 490 - Write Access Level 1/2
   // Write the acces level
   // 
   // DATA_ADDR: Modbus adr.: 412
   // DATA_LEN: 1 words
   // ENO of a box is taken as its EN; it also drops when the box reports an error
   #_w1 := #CMD_IN = 490;
   IF #_w1 THEN
       "MB_MASTER_DB"(REQ := #CMD_EN AND "MB_MASTER_DB".BUSY,   // MB_MASTER
                      MB_ADDR := #MB_ADDR,
                      MODE := 2,
                      DATA_ADDR := 40413,
                      DATA_LEN := 1,
                      DATA_PTR := #DB_PARA."Access level"."Access Password",
                      ERROR => #ERR_MB_MASTER,
                      STATUS => #STATUS_MB_MASTER);
       #CMD_EN := FALSE;
   END_IF;
   IF #_w1 AND "MB_MASTER_DB".DONE THEN #CMD_INPR_COUNT := 1; END_IF;
END_REGION

REGION Network 31: Command 490 - Write Access Level 2/2
   // Read the acces level to confirm new level
   // 
   // DATA_ADDR: Modbus adr.: 404
   // DATA_LEN: 1 words
   // ENO of a box is taken as its EN; it also drops when the box reports an error
   #_w1 := (#CMD_IN = 490) AND (#CMD_INPR_COUNT = 1);
   IF #_w1 THEN
       "MB_MASTER_DB"(REQ := "MB_MASTER_DB".BUSY,   // MB_MASTER
                      MB_ADDR := #MB_ADDR,
                      MODE := 2,
                      DATA_ADDR := 40405,
                      DATA_LEN := 1,
                      DATA_PTR := #DB_PARA."Access level"."Access level",
                      ERROR => #ERR_MB_MASTER,
                      STATUS => #STATUS_MB_MASTER);
   END_IF;
   IF #_w1 AND "MB_MASTER_DB".DONE THEN #CMD_INPR_COUNT := 0; END_IF;
END_REGION

REGION Network 32: Determine "CMD_INPR"
   RUNG wire#powerrail
      { S7_Templates := "SrcType := USInt" } GT_Contact(in1 := #CMD_INPR_COUNT, in2 := 0)
      wire#w1
      Coil( #CMD_INPR )
   END_RUNG
   RUNG wire#powerrail
      Contact( "MB_MASTER_DB".BUSY )
   END_RUNG wire#w1
   // the same network as SCL:
   #CMD_INPR := (#CMD_INPR_COUNT > 0) OR "MB_MASTER_DB".BUSY;
END_REGION

REGION Network 33: Check for Alarm/Error Status: Remove quality codes from alarm word (Bit 24 to bit 31)
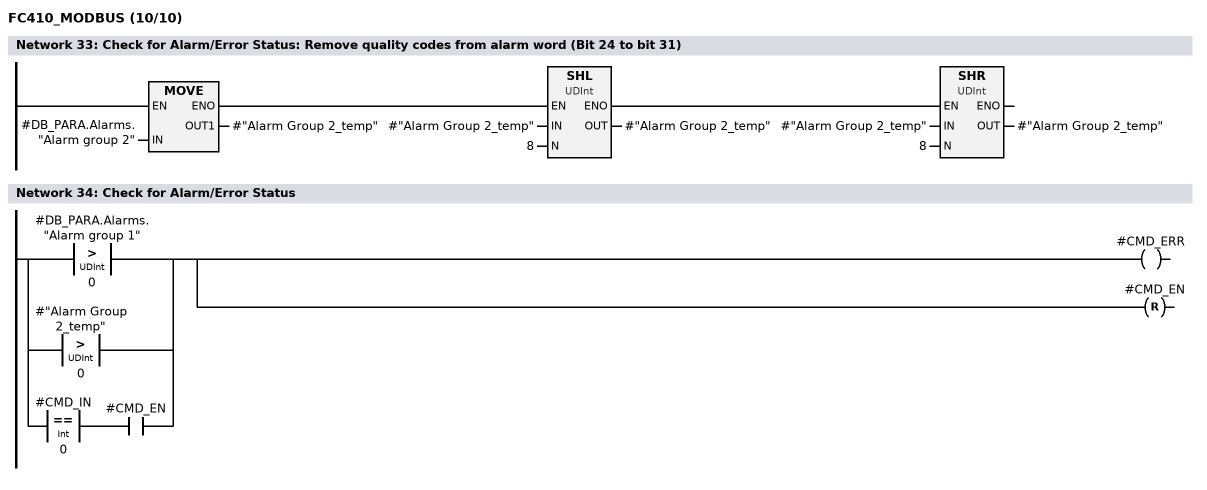
   RUNG wire#powerrail
      Move(in := #DB_PARA.Alarms."Alarm group 2", out1 => #"Alarm Group 2_temp")
      { S7_Templates := "SrcType := UDInt" } Shl(in := #"Alarm Group 2_temp", n := 8, out => #"Alarm Group 2_temp")
      { S7_Templates := "SrcType := UDInt" } Shr(in := #"Alarm Group 2_temp", n := 8, out => #"Alarm Group 2_temp")
   END_RUNG
   // the same network as SCL:
   #"Alarm Group 2_temp" := #DB_PARA.Alarms."Alarm group 2";
   #"Alarm Group 2_temp" := SHL(IN := #"Alarm Group 2_temp", N := 8);
   #"Alarm Group 2_temp" := SHR(IN := #"Alarm Group 2_temp", N := 8);
END_REGION

REGION Network 34: Check for Alarm/Error Status
   RUNG wire#powerrail
      { S7_Templates := "SrcType := UDInt" } GT_Contact(in1 := #DB_PARA.Alarms."Alarm group 1", in2 := 0)
      wire#w1
      Coil( #CMD_ERR )
   END_RUNG
   RUNG wire#powerrail
      { S7_Templates := "SrcType := UDInt" } GT_Contact(in1 := #"Alarm Group 2_temp", in2 := 0)
   END_RUNG wire#w1
   RUNG wire#powerrail
      { S7_Templates := "SrcType := Int" } EQ_Contact(in1 := #CMD_IN, in2 := 0)
      Contact( #CMD_EN )
   END_RUNG wire#w1
   RUNG wire#w1
      R_Coil( #CMD_EN )
   END_RUNG
   // the same network as SCL:
   #CMD_ERR := (#DB_PARA.Alarms."Alarm group 1" > 0) OR (#"Alarm Group 2_temp" > 0) OR ((#CMD_IN = 0) AND #CMD_EN);
   IF #CMD_ERR THEN #CMD_EN := FALSE; END_IF;
END_REGION
END_FUNCTION_BLOCK

FUNCTION_BLOCK "CONTADOR"   // FB2, LAD
{ S7_Optimized_Access := 'TRUE' }
VERSION : 0.1
   VAR_INPUT
      sSecadero : Bool;
      sHorno : Bool;
   END_VAR
   VAR_OUTPUT
      cSecadero : Int;
      cHorno : Int;
   END_VAR
BEGIN

REGION Network 1
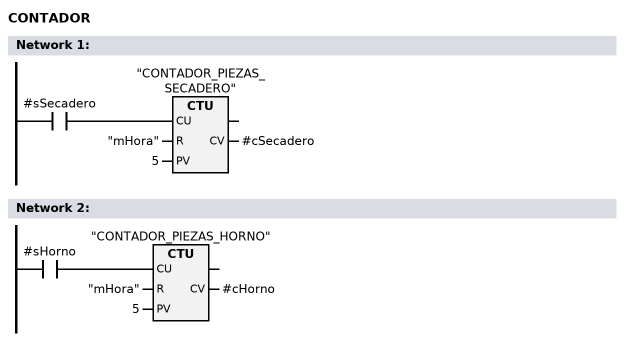
   "CONTADOR_PIEZAS_SECADERO".CTU(CU := #sSecadero, R := "mHora", PV := 5, CV => #cSecadero);
END_REGION

REGION Network 2
   "CONTADOR_PIEZAS_HORNO".CTU(CU := #sHorno, R := "mHora", PV := 5, CV => #cHorno);
END_REGION
END_FUNCTION_BLOCK

FUNCTION "FC410_INIT_MODBUS" : Void   // FC1, LAD
{ S7_Optimized_Access := 'TRUE' }
VERSION : 0.1
BEGIN

REGION Network 1: Comunicacion con MODBUS configuracion:
   // Default Modbus parameter from factory:
   // BAUDRATE: 19200
   // PARATY: EVEN => VALUE = 2
   // DATABITS: 8 bits
   // STOPBITS: 1 stopbit
   // PORT: 259 = from Device configuration ... CB1241
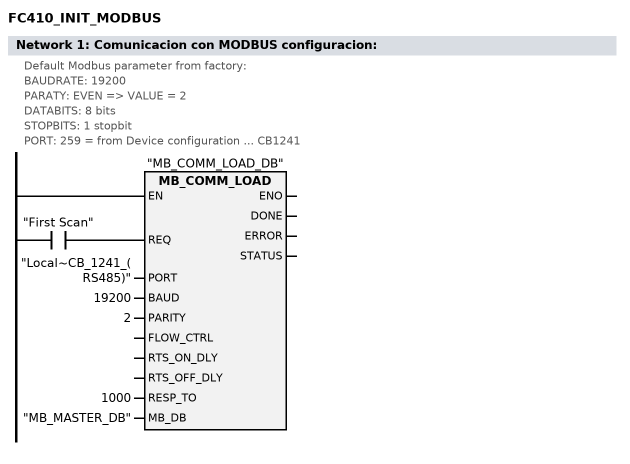
   "MB_COMM_LOAD_DB"(REQ := "First Scan",   // MB_COMM_LOAD
                     PORT := "Local~CB_1241_(RS485)",
                     BAUD := 19200,
                     PARITY := 2,
                     RESP_TO := 1000,
                     MB_DB := "MB_MASTER_DB");
END_REGION
END_FUNCTION

FUNCTION "FC410_DATA" : Void   // FC2, LAD
TITLE = Call of commands and FB for SITRANS FC410
{ S7_Optimized_Access := 'TRUE' }
VERSION : 0.1
   VAR_TEMP   // added for the SCL form of the ladder/FBD networks
      _w1 : Bool;
   END_VAR
BEGIN

REGION Network 1: Stop Read process values continiously: Command 200
   // Calling any other command will stop the continious read of process values
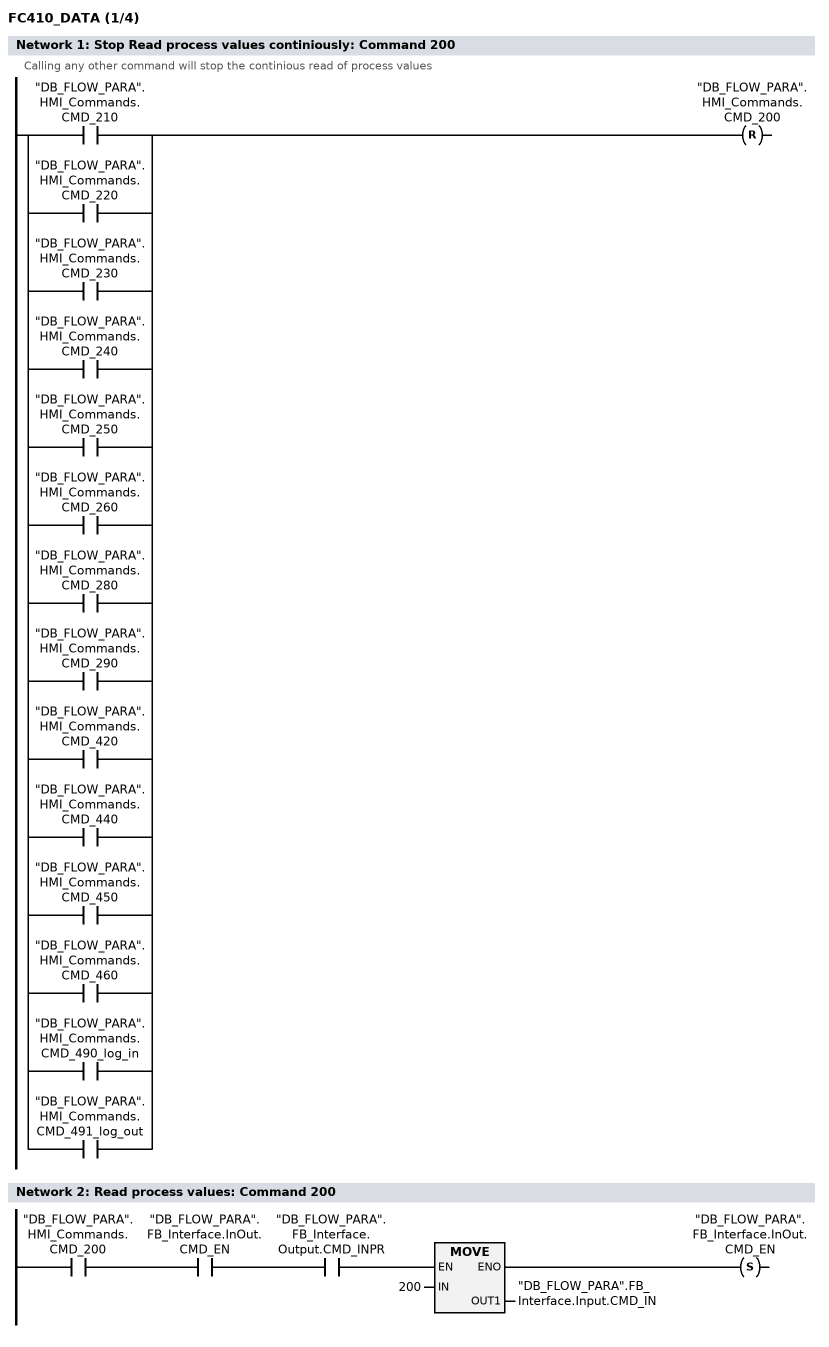
   RUNG wire#powerrail
      Contact( "DB_FLOW_PARA".HMI_Commands.CMD_210 )
      wire#w1
      R_Coil( "DB_FLOW_PARA".HMI_Commands.CMD_200 )
   END_RUNG
   RUNG wire#powerrail
      Contact( "DB_FLOW_PARA".HMI_Commands.CMD_220 )
   END_RUNG wire#w1
   RUNG wire#powerrail
      Contact( "DB_FLOW_PARA".HMI_Commands.CMD_230 )
   END_RUNG wire#w1
   RUNG wire#powerrail
      Contact( "DB_FLOW_PARA".HMI_Commands.CMD_240 )
   END_RUNG wire#w1
   RUNG wire#powerrail
      Contact( "DB_FLOW_PARA".HMI_Commands.CMD_250 )
   END_RUNG wire#w1
   RUNG wire#powerrail
      Contact( "DB_FLOW_PARA".HMI_Commands.CMD_260 )
   END_RUNG wire#w1
   RUNG wire#powerrail
      Contact( "DB_FLOW_PARA".HMI_Commands.CMD_280 )
   END_RUNG wire#w1
   RUNG wire#powerrail
      Contact( "DB_FLOW_PARA".HMI_Commands.CMD_290 )
   END_RUNG wire#w1
   RUNG wire#powerrail
      Contact( "DB_FLOW_PARA".HMI_Commands.CMD_420 )
   END_RUNG wire#w1
   RUNG wire#powerrail
      Contact( "DB_FLOW_PARA".HMI_Commands.CMD_440 )
   END_RUNG wire#w1
   RUNG wire#powerrail
      Contact( "DB_FLOW_PARA".HMI_Commands.CMD_450 )
   END_RUNG wire#w1
   RUNG wire#powerrail
      Contact( "DB_FLOW_PARA".HMI_Commands.CMD_460 )
   END_RUNG wire#w1
   RUNG wire#powerrail
      Contact( "DB_FLOW_PARA".HMI_Commands.CMD_490_log_in )
   END_RUNG wire#w1
   RUNG wire#powerrail
      Contact( "DB_FLOW_PARA".HMI_Commands.CMD_491_log_out )
   END_RUNG wire#w1
   // the same network as SCL:
   IF "DB_FLOW_PARA".HMI_Commands.CMD_210 OR "DB_FLOW_PARA".HMI_Commands.CMD_220 OR "DB_FLOW_PARA".HMI_Commands.CMD_230 OR "DB_FLOW_PARA".HMI_Commands.CMD_240 OR "DB_FLOW_PARA".HMI_Commands.CMD_250 OR "DB_FLOW_PARA".HMI_Commands.CMD_260 OR "DB_FLOW_PARA".HMI_Commands.CMD_280 OR "DB_FLOW_PARA".HMI_Commands.CMD_290 OR "DB_FLOW_PARA".HMI_Commands.CMD_420 OR "DB_FLOW_PARA".HMI_Commands.CMD_440 OR "DB_FLOW_PARA".HMI_Commands.CMD_450 OR "DB_FLOW_PARA".HMI_Commands.CMD_460 OR "DB_FLOW_PARA".HMI_Commands.CMD_490_log_in OR "DB_FLOW_PARA".HMI_Commands.CMD_491_log_out THEN
       "DB_FLOW_PARA".HMI_Commands.CMD_200 := FALSE;
   END_IF;
END_REGION

REGION Network 2: Read process values: Command 200
   RUNG wire#powerrail
      Contact( "DB_FLOW_PARA".HMI_Commands.CMD_200 )
      Contact( "DB_FLOW_PARA".FB_Interface.InOut.CMD_EN )
      Contact( "DB_FLOW_PARA".FB_Interface.Output.CMD_INPR )
      Move(in := 200, out1 => "DB_FLOW_PARA".FB_Interface.Input.CMD_IN)
      S_Coil( "DB_FLOW_PARA".FB_Interface.InOut.CMD_EN )
   END_RUNG
   // the same network as SCL:
   IF "DB_FLOW_PARA".HMI_Commands.CMD_200 AND "DB_FLOW_PARA".FB_Interface.InOut.CMD_EN AND "DB_FLOW_PARA".FB_Interface.Output.CMD_INPR THEN
       "DB_FLOW_PARA".FB_Interface.Input.CMD_IN := 200;
       "DB_FLOW_PARA".FB_Interface.InOut.CMD_EN := TRUE;
   END_IF;
END_REGION

REGION Network 3: Read identification data: Command 210
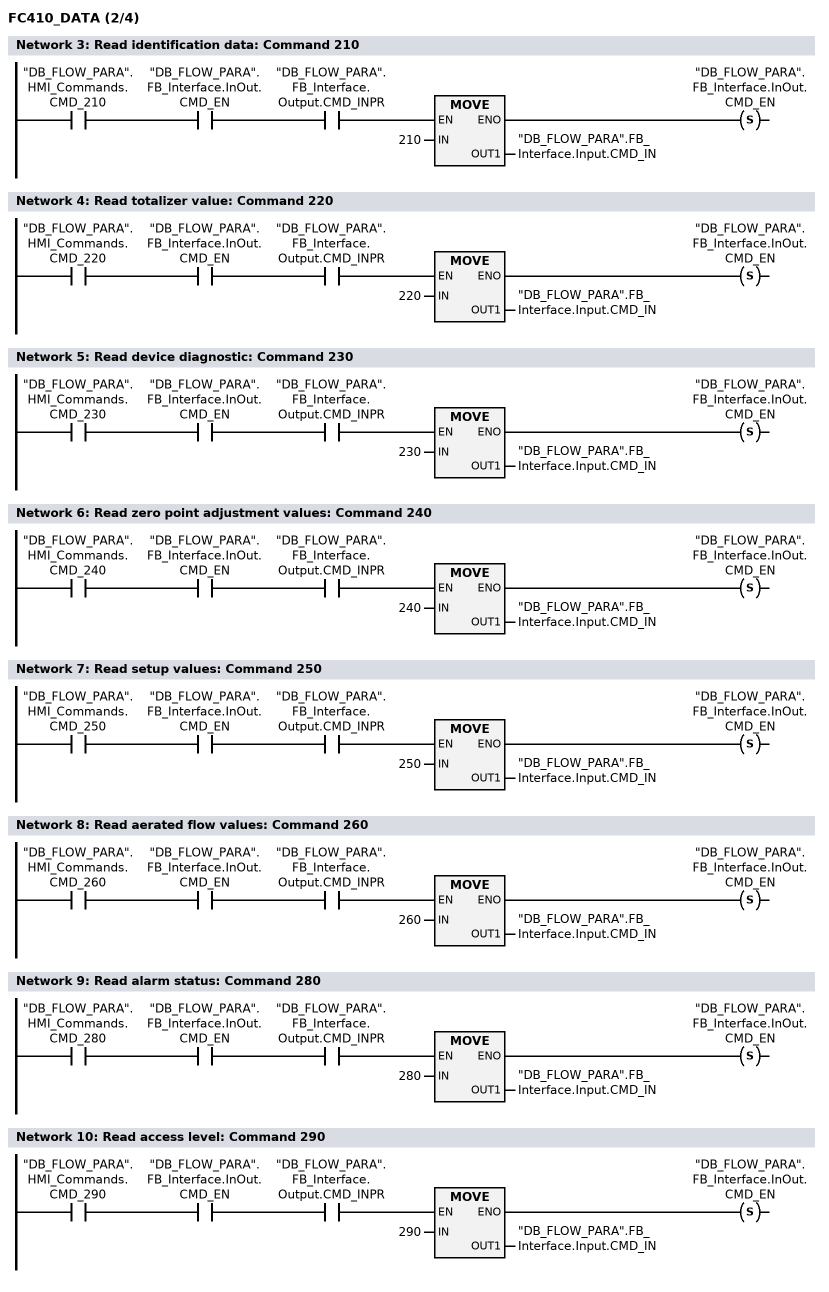
   RUNG wire#powerrail
      Contact( "DB_FLOW_PARA".HMI_Commands.CMD_210 )
      Contact( "DB_FLOW_PARA".FB_Interface.InOut.CMD_EN )
      Contact( "DB_FLOW_PARA".FB_Interface.Output.CMD_INPR )
      Move(in := 210, out1 => "DB_FLOW_PARA".FB_Interface.Input.CMD_IN)
      S_Coil( "DB_FLOW_PARA".FB_Interface.InOut.CMD_EN )
   END_RUNG
   // the same network as SCL:
   IF "DB_FLOW_PARA".HMI_Commands.CMD_210 AND "DB_FLOW_PARA".FB_Interface.InOut.CMD_EN AND "DB_FLOW_PARA".FB_Interface.Output.CMD_INPR THEN
       "DB_FLOW_PARA".FB_Interface.Input.CMD_IN := 210;
       "DB_FLOW_PARA".FB_Interface.InOut.CMD_EN := TRUE;
   END_IF;
END_REGION

REGION Network 4: Read totalizer value: Command 220
   RUNG wire#powerrail
      Contact( "DB_FLOW_PARA".HMI_Commands.CMD_220 )
      Contact( "DB_FLOW_PARA".FB_Interface.InOut.CMD_EN )
      Contact( "DB_FLOW_PARA".FB_Interface.Output.CMD_INPR )
      Move(in := 220, out1 => "DB_FLOW_PARA".FB_Interface.Input.CMD_IN)
      S_Coil( "DB_FLOW_PARA".FB_Interface.InOut.CMD_EN )
   END_RUNG
   // the same network as SCL:
   IF "DB_FLOW_PARA".HMI_Commands.CMD_220 AND "DB_FLOW_PARA".FB_Interface.InOut.CMD_EN AND "DB_FLOW_PARA".FB_Interface.Output.CMD_INPR THEN
       "DB_FLOW_PARA".FB_Interface.Input.CMD_IN := 220;
       "DB_FLOW_PARA".FB_Interface.InOut.CMD_EN := TRUE;
   END_IF;
END_REGION

REGION Network 5: Read device diagnostic: Command 230
   RUNG wire#powerrail
      Contact( "DB_FLOW_PARA".HMI_Commands.CMD_230 )
      Contact( "DB_FLOW_PARA".FB_Interface.InOut.CMD_EN )
      Contact( "DB_FLOW_PARA".FB_Interface.Output.CMD_INPR )
      Move(in := 230, out1 => "DB_FLOW_PARA".FB_Interface.Input.CMD_IN)
      S_Coil( "DB_FLOW_PARA".FB_Interface.InOut.CMD_EN )
   END_RUNG
   // the same network as SCL:
   IF "DB_FLOW_PARA".HMI_Commands.CMD_230 AND "DB_FLOW_PARA".FB_Interface.InOut.CMD_EN AND "DB_FLOW_PARA".FB_Interface.Output.CMD_INPR THEN
       "DB_FLOW_PARA".FB_Interface.Input.CMD_IN := 230;
       "DB_FLOW_PARA".FB_Interface.InOut.CMD_EN := TRUE;
   END_IF;
END_REGION

REGION Network 6: Read zero point adjustment values: Command 240
   RUNG wire#powerrail
      Contact( "DB_FLOW_PARA".HMI_Commands.CMD_240 )
      Contact( "DB_FLOW_PARA".FB_Interface.InOut.CMD_EN )
      Contact( "DB_FLOW_PARA".FB_Interface.Output.CMD_INPR )
      Move(in := 240, out1 => "DB_FLOW_PARA".FB_Interface.Input.CMD_IN)
      S_Coil( "DB_FLOW_PARA".FB_Interface.InOut.CMD_EN )
   END_RUNG
   // the same network as SCL:
   IF "DB_FLOW_PARA".HMI_Commands.CMD_240 AND "DB_FLOW_PARA".FB_Interface.InOut.CMD_EN AND "DB_FLOW_PARA".FB_Interface.Output.CMD_INPR THEN
       "DB_FLOW_PARA".FB_Interface.Input.CMD_IN := 240;
       "DB_FLOW_PARA".FB_Interface.InOut.CMD_EN := TRUE;
   END_IF;
END_REGION

REGION Network 7: Read setup values: Command 250
   RUNG wire#powerrail
      Contact( "DB_FLOW_PARA".HMI_Commands.CMD_250 )
      Contact( "DB_FLOW_PARA".FB_Interface.InOut.CMD_EN )
      Contact( "DB_FLOW_PARA".FB_Interface.Output.CMD_INPR )
      Move(in := 250, out1 => "DB_FLOW_PARA".FB_Interface.Input.CMD_IN)
      S_Coil( "DB_FLOW_PARA".FB_Interface.InOut.CMD_EN )
   END_RUNG
   // the same network as SCL:
   IF "DB_FLOW_PARA".HMI_Commands.CMD_250 AND "DB_FLOW_PARA".FB_Interface.InOut.CMD_EN AND "DB_FLOW_PARA".FB_Interface.Output.CMD_INPR THEN
       "DB_FLOW_PARA".FB_Interface.Input.CMD_IN := 250;
       "DB_FLOW_PARA".FB_Interface.InOut.CMD_EN := TRUE;
   END_IF;
END_REGION

REGION Network 8: Read aerated flow values: Command 260
   RUNG wire#powerrail
      Contact( "DB_FLOW_PARA".HMI_Commands.CMD_260 )
      Contact( "DB_FLOW_PARA".FB_Interface.InOut.CMD_EN )
      Contact( "DB_FLOW_PARA".FB_Interface.Output.CMD_INPR )
      Move(in := 260, out1 => "DB_FLOW_PARA".FB_Interface.Input.CMD_IN)
      S_Coil( "DB_FLOW_PARA".FB_Interface.InOut.CMD_EN )
   END_RUNG
   // the same network as SCL:
   IF "DB_FLOW_PARA".HMI_Commands.CMD_260 AND "DB_FLOW_PARA".FB_Interface.InOut.CMD_EN AND "DB_FLOW_PARA".FB_Interface.Output.CMD_INPR THEN
       "DB_FLOW_PARA".FB_Interface.Input.CMD_IN := 260;
       "DB_FLOW_PARA".FB_Interface.InOut.CMD_EN := TRUE;
   END_IF;
END_REGION

REGION Network 9: Read alarm status: Command 280
   RUNG wire#powerrail
      Contact( "DB_FLOW_PARA".HMI_Commands.CMD_280 )
      Contact( "DB_FLOW_PARA".FB_Interface.InOut.CMD_EN )
      Contact( "DB_FLOW_PARA".FB_Interface.Output.CMD_INPR )
      Move(in := 280, out1 => "DB_FLOW_PARA".FB_Interface.Input.CMD_IN)
      S_Coil( "DB_FLOW_PARA".FB_Interface.InOut.CMD_EN )
   END_RUNG
   // the same network as SCL:
   IF "DB_FLOW_PARA".HMI_Commands.CMD_280 AND "DB_FLOW_PARA".FB_Interface.InOut.CMD_EN AND "DB_FLOW_PARA".FB_Interface.Output.CMD_INPR THEN
       "DB_FLOW_PARA".FB_Interface.Input.CMD_IN := 280;
       "DB_FLOW_PARA".FB_Interface.InOut.CMD_EN := TRUE;
   END_IF;
END_REGION

REGION Network 10: Read access level: Command 290
   RUNG wire#powerrail
      Contact( "DB_FLOW_PARA".HMI_Commands.CMD_290 )
      Contact( "DB_FLOW_PARA".FB_Interface.InOut.CMD_EN )
      Contact( "DB_FLOW_PARA".FB_Interface.Output.CMD_INPR )
      Move(in := 290, out1 => "DB_FLOW_PARA".FB_Interface.Input.CMD_IN)
      S_Coil( "DB_FLOW_PARA".FB_Interface.InOut.CMD_EN )
   END_RUNG
   // the same network as SCL:
   IF "DB_FLOW_PARA".HMI_Commands.CMD_290 AND "DB_FLOW_PARA".FB_Interface.InOut.CMD_EN AND "DB_FLOW_PARA".FB_Interface.Output.CMD_INPR THEN
       "DB_FLOW_PARA".FB_Interface.Input.CMD_IN := 290;
       "DB_FLOW_PARA".FB_Interface.InOut.CMD_EN := TRUE;
   END_IF;
END_REGION

REGION Network 11: Write, reset totalizer: Command 420
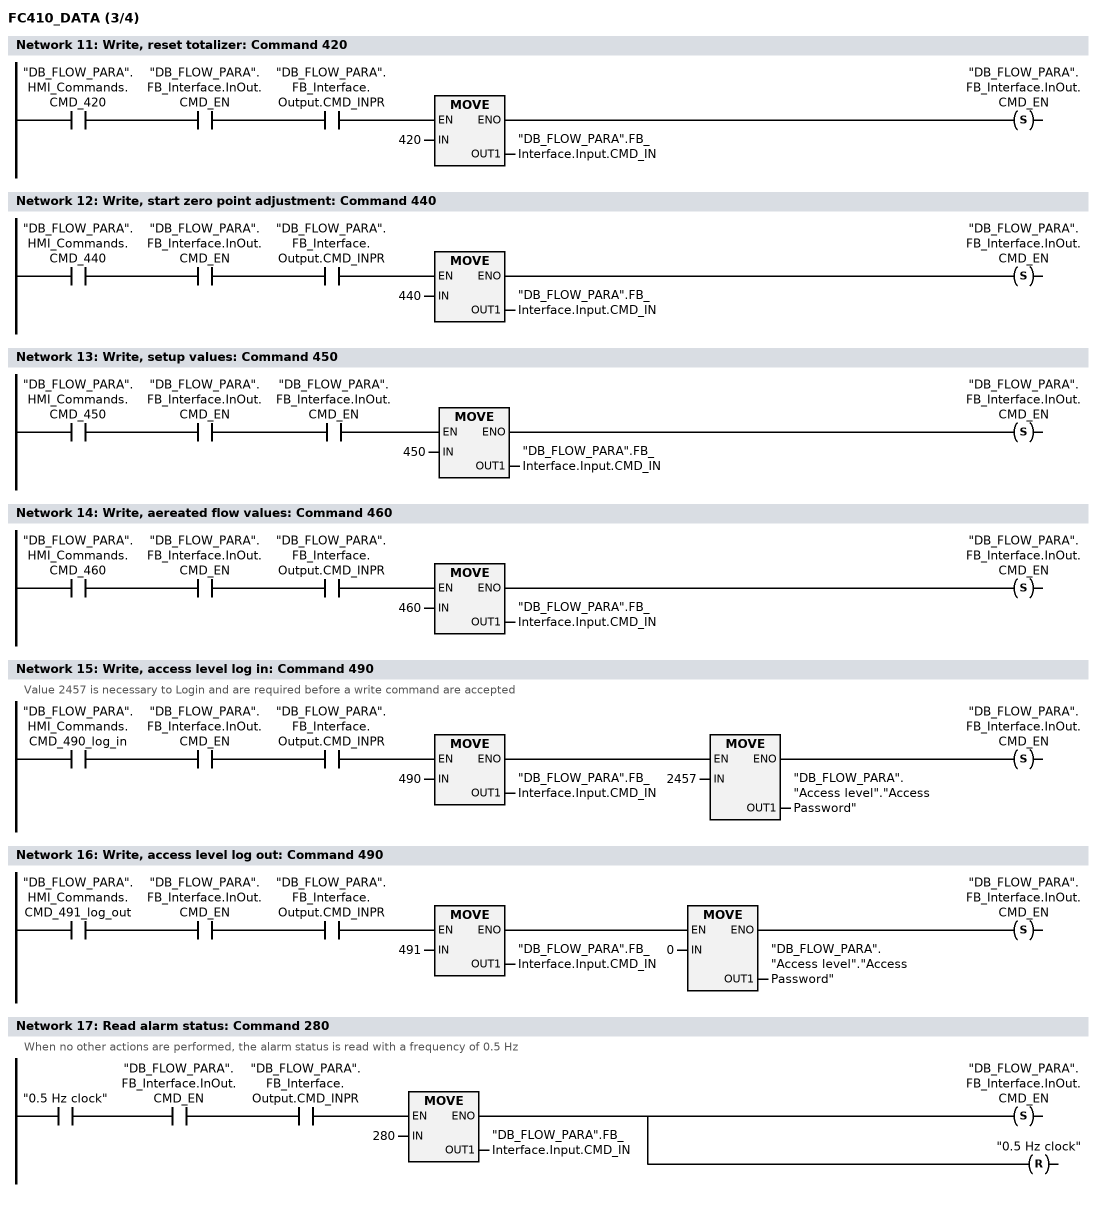
   RUNG wire#powerrail
      Contact( "DB_FLOW_PARA".HMI_Commands.CMD_420 )
      Contact( "DB_FLOW_PARA".FB_Interface.InOut.CMD_EN )
      Contact( "DB_FLOW_PARA".FB_Interface.Output.CMD_INPR )
      Move(in := 420, out1 => "DB_FLOW_PARA".FB_Interface.Input.CMD_IN)
      S_Coil( "DB_FLOW_PARA".FB_Interface.InOut.CMD_EN )
   END_RUNG
   // the same network as SCL:
   IF "DB_FLOW_PARA".HMI_Commands.CMD_420 AND "DB_FLOW_PARA".FB_Interface.InOut.CMD_EN AND "DB_FLOW_PARA".FB_Interface.Output.CMD_INPR THEN
       "DB_FLOW_PARA".FB_Interface.Input.CMD_IN := 420;
       "DB_FLOW_PARA".FB_Interface.InOut.CMD_EN := TRUE;
   END_IF;
END_REGION

REGION Network 12: Write, start zero point adjustment: Command 440
   RUNG wire#powerrail
      Contact( "DB_FLOW_PARA".HMI_Commands.CMD_440 )
      Contact( "DB_FLOW_PARA".FB_Interface.InOut.CMD_EN )
      Contact( "DB_FLOW_PARA".FB_Interface.Output.CMD_INPR )
      Move(in := 440, out1 => "DB_FLOW_PARA".FB_Interface.Input.CMD_IN)
      S_Coil( "DB_FLOW_PARA".FB_Interface.InOut.CMD_EN )
   END_RUNG
   // the same network as SCL:
   IF "DB_FLOW_PARA".HMI_Commands.CMD_440 AND "DB_FLOW_PARA".FB_Interface.InOut.CMD_EN AND "DB_FLOW_PARA".FB_Interface.Output.CMD_INPR THEN
       "DB_FLOW_PARA".FB_Interface.Input.CMD_IN := 440;
       "DB_FLOW_PARA".FB_Interface.InOut.CMD_EN := TRUE;
   END_IF;
END_REGION

REGION Network 13: Write, setup values: Command 450
   RUNG wire#powerrail
      Contact( "DB_FLOW_PARA".HMI_Commands.CMD_450 )
      Contact( "DB_FLOW_PARA".FB_Interface.InOut.CMD_EN )
      Contact( "DB_FLOW_PARA".FB_Interface.InOut.CMD_EN )
      Move(in := 450, out1 => "DB_FLOW_PARA".FB_Interface.Input.CMD_IN)
      S_Coil( "DB_FLOW_PARA".FB_Interface.InOut.CMD_EN )
   END_RUNG
   // the same network as SCL:
   IF "DB_FLOW_PARA".HMI_Commands.CMD_450 AND "DB_FLOW_PARA".FB_Interface.InOut.CMD_EN AND "DB_FLOW_PARA".FB_Interface.InOut.CMD_EN THEN
       "DB_FLOW_PARA".FB_Interface.Input.CMD_IN := 450;
       "DB_FLOW_PARA".FB_Interface.InOut.CMD_EN := TRUE;
   END_IF;
END_REGION

REGION Network 14: Write, aereated flow values: Command 460
   RUNG wire#powerrail
      Contact( "DB_FLOW_PARA".HMI_Commands.CMD_460 )
      Contact( "DB_FLOW_PARA".FB_Interface.InOut.CMD_EN )
      Contact( "DB_FLOW_PARA".FB_Interface.Output.CMD_INPR )
      Move(in := 460, out1 => "DB_FLOW_PARA".FB_Interface.Input.CMD_IN)
      S_Coil( "DB_FLOW_PARA".FB_Interface.InOut.CMD_EN )
   END_RUNG
   // the same network as SCL:
   IF "DB_FLOW_PARA".HMI_Commands.CMD_460 AND "DB_FLOW_PARA".FB_Interface.InOut.CMD_EN AND "DB_FLOW_PARA".FB_Interface.Output.CMD_INPR THEN
       "DB_FLOW_PARA".FB_Interface.Input.CMD_IN := 460;
       "DB_FLOW_PARA".FB_Interface.InOut.CMD_EN := TRUE;
   END_IF;
END_REGION

REGION Network 15: Write, access level log in: Command 490
   // Value 2457 is necessary to Login and are required before a write command are accepted
   RUNG wire#powerrail
      Contact( "DB_FLOW_PARA".HMI_Commands.CMD_490_log_in )
      Contact( "DB_FLOW_PARA".FB_Interface.InOut.CMD_EN )
      Contact( "DB_FLOW_PARA".FB_Interface.Output.CMD_INPR )
      Move(in := 490, out1 => "DB_FLOW_PARA".FB_Interface.Input.CMD_IN)
      Move(in := 2457, out1 => "DB_FLOW_PARA"."Access level"."Access Password")
      S_Coil( "DB_FLOW_PARA".FB_Interface.InOut.CMD_EN )
   END_RUNG
   // the same network as SCL:
   IF "DB_FLOW_PARA".HMI_Commands.CMD_490_log_in AND "DB_FLOW_PARA".FB_Interface.InOut.CMD_EN AND "DB_FLOW_PARA".FB_Interface.Output.CMD_INPR THEN
       "DB_FLOW_PARA".FB_Interface.Input.CMD_IN := 490;
       "DB_FLOW_PARA"."Access level"."Access Password" := 2457;
       "DB_FLOW_PARA".FB_Interface.InOut.CMD_EN := TRUE;
   END_IF;
END_REGION

REGION Network 16: Write, access level log out: Command 490
   RUNG wire#powerrail
      Contact( "DB_FLOW_PARA".HMI_Commands.CMD_491_log_out )
      Contact( "DB_FLOW_PARA".FB_Interface.InOut.CMD_EN )
      Contact( "DB_FLOW_PARA".FB_Interface.Output.CMD_INPR )
      Move(in := 491, out1 => "DB_FLOW_PARA".FB_Interface.Input.CMD_IN)
      Move(in := 0, out1 => "DB_FLOW_PARA"."Access level"."Access Password")
      S_Coil( "DB_FLOW_PARA".FB_Interface.InOut.CMD_EN )
   END_RUNG
   // the same network as SCL:
   IF "DB_FLOW_PARA".HMI_Commands.CMD_491_log_out AND "DB_FLOW_PARA".FB_Interface.InOut.CMD_EN AND "DB_FLOW_PARA".FB_Interface.Output.CMD_INPR THEN
       "DB_FLOW_PARA".FB_Interface.Input.CMD_IN := 491;
       "DB_FLOW_PARA"."Access level"."Access Password" := 0;
       "DB_FLOW_PARA".FB_Interface.InOut.CMD_EN := TRUE;
   END_IF;
END_REGION

REGION Network 17: Read alarm status: Command 280
   // When no other actions are performed, the alarm status is read with a frequency of 0.5 Hz
   RUNG wire#powerrail
      Contact( "0.5 Hz clock" )
      Contact( "DB_FLOW_PARA".FB_Interface.InOut.CMD_EN )
      Contact( "DB_FLOW_PARA".FB_Interface.Output.CMD_INPR )
      Move(in := 280, out1 => "DB_FLOW_PARA".FB_Interface.Input.CMD_IN)
      wire#w1
      S_Coil( "DB_FLOW_PARA".FB_Interface.InOut.CMD_EN )
   END_RUNG
   RUNG wire#w1
      R_Coil( "0.5 Hz clock" )
   END_RUNG
   // the same network as SCL:
   IF "0.5 Hz clock" AND "DB_FLOW_PARA".FB_Interface.InOut.CMD_EN AND "DB_FLOW_PARA".FB_Interface.Output.CMD_INPR THEN
       "DB_FLOW_PARA".FB_Interface.Input.CMD_IN := 280;
   END_IF;
   #_w1 := "0.5 Hz clock" AND "DB_FLOW_PARA".FB_Interface.InOut.CMD_EN AND "DB_FLOW_PARA".FB_Interface.Output.CMD_INPR;
   IF #_w1 THEN
       "DB_FLOW_PARA".FB_Interface.InOut.CMD_EN := TRUE;
       "0.5 Hz clock" := FALSE;
   END_IF;
END_REGION

REGION Network 18: Set Modbus address
   // Default factory Modbus address is: 1
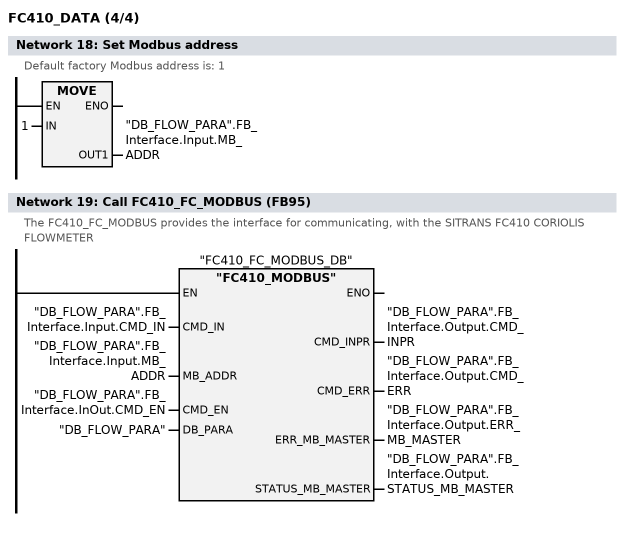
   RUNG wire#powerrail
      Move(in := 1, out1 => "DB_FLOW_PARA".FB_Interface.Input.MB_ADDR)
   END_RUNG
   // the same network as SCL:
   "DB_FLOW_PARA".FB_Interface.Input.MB_ADDR := 1;
END_REGION

REGION Network 19: Call FC410_FC_MODBUS (FB95)
   // The FC410_FC_MODBUS provides the interface for communicating, with the SITRANS FC410 CORIOLIS FLOWMETER
   RUNG wire#powerrail
      "FC410_FC_MODBUS_DB"(CMD_IN := "DB_FLOW_PARA".FB_Interface.Input.CMD_IN, MB_ADDR := "DB_FLOW_PARA".FB_Interface.Input.MB_ADDR, CMD_EN := "DB_FLOW_PARA".FB_Interface.InOut.CMD_EN, DB_PARA := "DB_FLOW_PARA", CMD_INPR => "DB_FLOW_PARA".FB_Interface.Output.CMD_INPR, CMD_ERR => "DB_FLOW_PARA".FB_Interface.Output.CMD_ERR, ERR_MB_MASTER => "DB_FLOW_PARA".FB_Interface.Output.ERR_MB_MASTER, STATUS_MB_MASTER => "DB_FLOW_PARA".FB_Interface.Output.STATUS_MB_MASTER)
   END_RUNG
   // the same network as SCL:
   "FC410_FC_MODBUS_DB"(CMD_IN := "DB_FLOW_PARA".FB_Interface.Input.CMD_IN,   // "FC410_MODBUS"
                        MB_ADDR := "DB_FLOW_PARA".FB_Interface.Input.MB_ADDR,
                        CMD_EN := "DB_FLOW_PARA".FB_Interface.InOut.CMD_EN,
                        DB_PARA := "DB_FLOW_PARA",
                        CMD_INPR => "DB_FLOW_PARA".FB_Interface.Output.CMD_INPR,
                        CMD_ERR => "DB_FLOW_PARA".FB_Interface.Output.CMD_ERR,
                        ERR_MB_MASTER => "DB_FLOW_PARA".FB_Interface.Output.ERR_MB_MASTER,
                        STATUS_MB_MASTER => "DB_FLOW_PARA".FB_Interface.Output.STATUS_MB_MASTER);
END_REGION
END_FUNCTION

FUNCTION "RESET_CONTADOR" : Void   // FC3, LAD
{ S7_Optimized_Access := 'TRUE' }
VERSION : 0.1
   VAR_OUTPUT
      m_hora : Int;
      reset_c : Bool;
   END_VAR
BEGIN

REGION Network 1
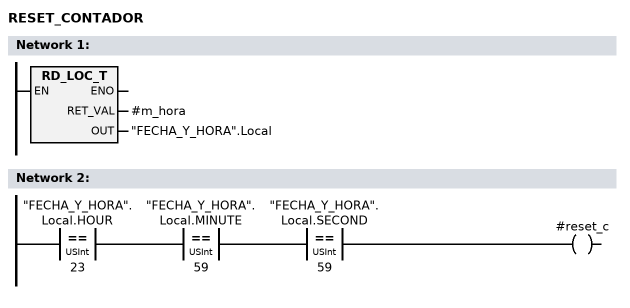
   #m_hora := RD_LOC_T(OUT => "FECHA_Y_HORA".Local);
END_REGION

REGION Network 2
   RUNG wire#powerrail
      { S7_Templates := "SrcType := USInt" } EQ_Contact(in1 := "FECHA_Y_HORA".Local.HOUR, in2 := 23)
      { S7_Templates := "SrcType := USInt" } EQ_Contact(in1 := "FECHA_Y_HORA".Local.MINUTE, in2 := 59)
      { S7_Templates := "SrcType := USInt" } EQ_Contact(in1 := "FECHA_Y_HORA".Local.SECOND, in2 := 59)
      Coil( #reset_c )
   END_RUNG
   // the same network as SCL:
   #reset_c := ("FECHA_Y_HORA".Local.HOUR = 23) AND ("FECHA_Y_HORA".Local.MINUTE = 59) AND ("FECHA_Y_HORA".Local.SECOND = 59);
END_REGION
END_FUNCTION

ORGANIZATION_BLOCK "Main"   // OB1, LAD, ProgramCycle
TITLE = "Main Program Sweep (Cycle)"
{ S7_Optimized_Access := 'TRUE' }
VERSION : 0.1
   VAR_INPUT
      Initial_Call : Bool;   // Initial call of this OB
      Remanence : Bool;   // =True, if remanent data are available
   END_VAR
BEGIN

REGION Network 1
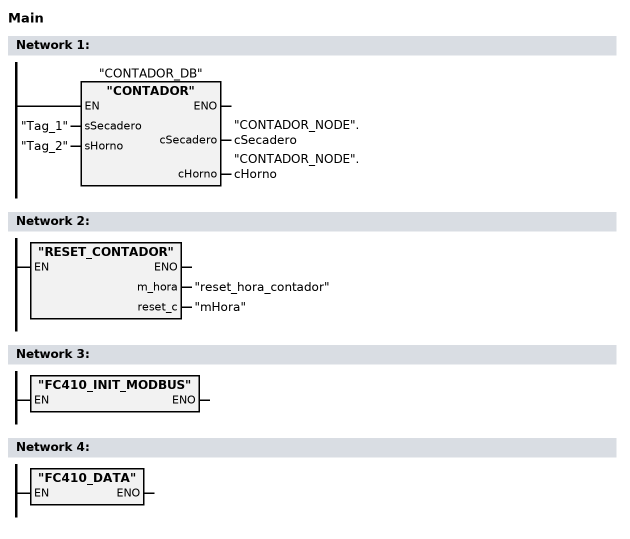
   RUNG wire#powerrail
      "CONTADOR_DB"(sSecadero := "Tag_1", sHorno := "Tag_2", cSecadero => "CONTADOR_NODE".cSecadero, cHorno => "CONTADOR_NODE".cHorno)
   END_RUNG
   // the same network as SCL:
   "CONTADOR_DB"(sSecadero := "Tag_1",   // "CONTADOR"
                 sHorno := "Tag_2",
                 cSecadero => "CONTADOR_NODE".cSecadero,
                 cHorno => "CONTADOR_NODE".cHorno);
END_REGION

REGION Network 2
   RUNG wire#powerrail
      "RESET_CONTADOR"(m_hora => "reset_hora_contador", reset_c => "mHora")
   END_RUNG
   // the same network as SCL:
   "RESET_CONTADOR"(m_hora => "reset_hora_contador", reset_c => "mHora");
END_REGION

REGION Network 3
   RUNG wire#powerrail
      "FC410_INIT_MODBUS"()
   END_RUNG
   // the same network as SCL:
   "FC410_INIT_MODBUS"();
END_REGION

REGION Network 4
   RUNG wire#powerrail
      "FC410_DATA"()
   END_RUNG
   // the same network as SCL:
   "FC410_DATA"();
END_REGION
END_ORGANIZATION_BLOCK

(* ===== HMI "HMI_RT_1" =====
system functions are stored by id; their names below are inferred from use
connection "HMI_Conexión_1": ETHERNET, SMART_S7_1200_OMS

HMI tags "Tabla de variables estándar"
   "DB_FLOW_PARA_Access level.Access level" : UInt = PLC DB_FLOW_PARA."Access level"."Access level" AT %DB17.DBW116, 1 s
   "DB_FLOW_PARA_HMI_Commands.CMD_290" : Bool = PLC DB_FLOW_PARA.HMI_Commands.CMD_290 AT %DB17.DBX121.0, 1 s
   "DB_FLOW_PARA_Setup.Low Massflow cutofff" : Real = PLC DB_FLOW_PARA.Setup."Low Massflow cutofff" AT %DB17.DBD84, 1 s
   "DB_FLOW_PARA_Setup.Low volumeflow cutoff" : Real = PLC DB_FLOW_PARA.Setup."Low volumeflow cutoff" AT %DB17.DBD88, 1 s
   "DB_FLOW_PARA_Setup.Process noise damping" : UInt = PLC DB_FLOW_PARA.Setup."Process noise damping" AT %DB17.DBW82, 1 s
   "DB_FLOW_PARA_Setup.Flow direction" : UInt = PLC DB_FLOW_PARA.Setup."Flow direction" AT %DB17.DBW80, 1 s
   "DB_FLOW_PARA_HMI_Commands.CMD_250" : Bool = PLC DB_FLOW_PARA.HMI_Commands.CMD_250 AT %DB17.DBX120.5, 1 s
   "DB_FLOW_PARA_HMI_Commands.CMD_450" : Bool = PLC DB_FLOW_PARA.HMI_Commands.CMD_450 AT %DB17.DBX121.3, 1 s
   "DB_FLOW_PARA_Zero Point adjustment.Zero point duration" : UInt = PLC DB_FLOW_PARA."Zero Point adjustment"."Zero point duration" AT %DB17.DBW64, 1 s
   "DB_FLOW_PARA_Zero Point adjustment.Zero point offset value" : Real = PLC DB_FLOW_PARA."Zero Point adjustment"."Zero point offset value" AT %DB17.DBD70, 1 s
   "DB_FLOW_PARA_Zero Point adjustment.Standard deviation" : Real = PLC DB_FLOW_PARA."Zero Point adjustment"."Standard deviation" AT %DB17.DBD66, 1 s
   "DB_FLOW_PARA_Zero Point adjustment.Zero point adjust progress" : UInt = PLC DB_FLOW_PARA."Zero Point adjustment"."Zero point adjust progress" AT %DB17.DBW74, 1 s
   "DB_FLOW_PARA_HMI_Commands.CMD_240" : Bool = PLC DB_FLOW_PARA.HMI_Commands.CMD_240 AT %DB17.DBX120.4, 1 s
   "DB_FLOW_PARA_HMI_Commands.CMD_440" : Bool = PLC DB_FLOW_PARA.HMI_Commands.CMD_440 AT %DB17.DBX121.2, 1 s
   "DB_FLOW_PARA_Totalizer.Totalizer value" : Real = PLC DB_FLOW_PARA.Totalizer."Totalizer value" AT %DB17.DBD42, 1 s
   "DB_FLOW_PARA_HMI_Commands.CMD_220" : Bool = PLC DB_FLOW_PARA.HMI_Commands.CMD_220 AT %DB17.DBX120.2, 1 s
   "DB_FLOW_PARA_HMI_Commands.CMD_420" : Bool = PLC DB_FLOW_PARA.HMI_Commands.CMD_420 AT %DB17.DBX121.1, 1 s
   "DB_FLOW_PARA_Identification data.Sensor serial number" : String[20] = PLC DB_FLOW_PARA."Identification data"."Sensor serial number" AT %DB17.DBX20.0, 1 s
   "DB_FLOW_PARA_HMI_Commands.CMD_210" : Bool = PLC DB_FLOW_PARA.HMI_Commands.CMD_210 AT %DB17.DBX120.1, 1 s
   "DB_FLOW_PARA_Process Values.Massflow" : Real = PLC DB_FLOW_PARA."Process Values".Massflow AT %DB17.DBD0, 1 s
   "DB_FLOW_PARA_Process Values.Volumeflow" : Real = PLC DB_FLOW_PARA."Process Values".Volumeflow AT %DB17.DBD4, 1 s
   "DB_FLOW_PARA_Process Values.Density" : Real = PLC DB_FLOW_PARA."Process Values".Density AT %DB17.DBD8, 1 s
   "DB_FLOW_PARA_Process Values.Temperature" : Real = PLC DB_FLOW_PARA."Process Values".Temperature AT %DB17.DBD12, 1 s
   "DB_FLOW_PARA_Process Values.Frame temperature" : Real = PLC DB_FLOW_PARA."Process Values"."Frame temperature" AT %DB17.DBD16, 1 s
   "DB_FLOW_PARA_HMI_Commands.CMD_200" : Bool = PLC DB_FLOW_PARA.HMI_Commands.CMD_200 AT %DB17.DBX120.0, 1 s
   "DB_FLOW_PARA_HMI_Commands.CMD_490_log_in" : Bool = PLC DB_FLOW_PARA.HMI_Commands.CMD_490_log_in AT %DB17.DBX121.5, 1 s
   "DB_FLOW_PARA_HMI_Commands.CMD_491_log_out" : Bool = PLC DB_FLOW_PARA.HMI_Commands.CMD_491_log_out AT %DB17.DBX121.6, 1 s
   "DB_FLOW_PARA_HMI_Commands.CMD_230" : Bool = PLC DB_FLOW_PARA.HMI_Commands.CMD_230 AT %DB17.DBX120.3, 1 s
   "DB_FLOW_PARA_HMI_Commands.CMD_280" : Bool = PLC DB_FLOW_PARA.HMI_Commands.CMD_280 AT %DB17.DBX120.7, 1 s
   "DB_FLOW_PARA_Alarms.Alarm group 1" : UDInt = PLC DB_FLOW_PARA.Alarms."Alarm group 1" AT %DB17.DBD108, 1 s
   "DB_FLOW_PARA_Alarms.Alarm group 2" : UDInt = PLC DB_FLOW_PARA.Alarms."Alarm group 2" AT %DB17.DBD112, 1 s
   "CONTADOR_DB_cHorno" : Int = PLC CONTADOR_DB.cHorno, 1 s
   "CONTADOR_DB_cSecadero" : Int = PLC CONTADOR_DB.cSecadero, 1 s

text list "Access level": 4 '04: Logged Out'; 16 '16: Logged Out'; 32 '32: Logged In'

text list "Process Noise Damping": 0 '0: 55 ms filtering (Centrifugal Pump)'; 1 '1: 110 ms filtering (Triplex Pump)'; 2 '2: 220 ms filtering (Duples Pump)'; 3 '3: 400 ms filtering (Simplex Pump)'; 4 '4: 800 ms filtering (Cam Pump)'

text list "Flow direction": 0 '0: Negative'; 1 '1: Positive'

Template "Plantilla_1" 320x240
   Button "Salir" at 266,202 size 52x37; TextOff 'Salir'; PictureOff "ExitRuntime_KTP600_Basic_color_PN"; PictureOn "ExitRuntime_KTP600_Basic_color_PN"
      on Release: StopRuntime(0)
   Button "Template_Button" at 213,202 size 52x37; TextOff 'Text'
   Button "Template_Button_1" at 160,202 size 52x37; TextOff 'Text'
   Button "Template_Button_2" at 107,202 size 52x37; TextOff 'Text'
   Button "Template_Button_3" at 54,202 size 52x37; TextOff 'Text'
   Button "Imagen inicial" at 1,202 size 52x37; TextOff 'Imagen inicial'; PictureOff "NavigateHome_KTP600_Basic_color_PN"; PictureOn "NavigateHome_KTP600_Basic_color_PN"
      on Release: ActivateScreen("Imagen raíz", 0)

screen "Imagen raíz" 320x240, template "Plantilla_1"
   Button "Botón_1" at 52,202 size 52x37; TextOff 'Configu- racion'
      on Click: ActivateScreen("101_Access_Level", 0)
   Button "Botón_2" at 104,202 size 56x37; TextOff 'Identi- ficacion'
      on Click: ActivateScreen("200_Identification", 0)
   Button "Botón_3" at 160,202 size 55x37; TextOff 'Operating'
      on Click: ActivateScreen("300_Operating", 0)
   Button "Botón_4" at 213,202 size 54x37; TextOff 'Diag- nostico'
      on Click: ActivateScreen("400_Diagnose", 0)

screen "101_Access_Level" 320x240, template "Plantilla_1"
   Button "Botón_1" at 106,202 size 52x37; TextOff 'Read'
      on Press: SetBit("DB_FLOW_PARA_HMI_Commands.CMD_290")
      on Release: ResetBit("DB_FLOW_PARA_HMI_Commands.CMD_290")
   Button "Botón_2" at 159,202 size 53x37; TextOff 'Log In'
      on Release: ResetBit("DB_FLOW_PARA_HMI_Commands.CMD_490_log_in"); ActivateScreen("100_Setup", 0)
      on Press: SetBit("DB_FLOW_PARA_HMI_Commands.CMD_490_log_in")
   Button "Botón_3" at 212,202 size 53x37; TextOff 'Log Out'
      on Release: ResetBit("DB_FLOW_PARA_HMI_Commands.CMD_491_log_out"); ActivateScreen("Imagen raíz", 0)
      on Press: SetBit("DB_FLOW_PARA_HMI_Commands.CMD_491_log_out")
   TextField "Campo de texto_2" at 26,53 size 86x16; Text 'Nivel de acceso'
   SymbolicIOField "Campo ES simbólico_2" at 147,52 size 129x17; TextOn '1'; TextOff '0'; TextList "Access level"
      ProcessValue <- "DB_FLOW_PARA_Access level.Access level"
   TextField "Campo de texto_7" at 124,4 size 93x16; Text 'Nivel de acceso'

screen "100_Setup" 320x240, template "Plantilla_1"
   Button "Botón_1" at 86,27 size 135x32; TextOff 'Configuracion de flujo'
      on Click: ActivateScreen("110_Flow_Setup", 0)
   Button "Botón_2" at 87,66 size 134x32; TextOff 'Ajuste punto cero'
      on Release: ActivateScreen("120_Zero_Point_Adjust", 0)
   Button "Botón_3" at 85,108 size 136x32; TextOff 'Flujo aireado'
      on Click: ActivateScreen("131_Aerated_Flow", 0)
   Button "Botón_4" at 85,150 size 135x32; TextOff 'Totalizador'
      on Click: ActivateScreen("140_Totalizer", 0)

screen "110_Flow_Setup" 320x240, template "Plantilla_1"
   Button "Botón_1" at 54,203 size 52x36; TextOff 'Setup'
      on Click: ActivateScreen("100_Setup", 0)
   Button "Botón_2" at 160,203 size 52x36; TextOff 'Read'
      on Press: SetBit("DB_FLOW_PARA_HMI_Commands.CMD_250")
      on Release: ResetBit("DB_FLOW_PARA_HMI_Commands.CMD_250")
   Button "Botón_3" at 214,203 size 51x36; TextOff 'Write'
      on Press: SetBit("DB_FLOW_PARA_HMI_Commands.CMD_450")
      on Release: ResetBit("DB_FLOW_PARA_HMI_Commands.CMD_450")
   TextField "Campo de texto_7" at 124,4 size 87x16; Text 'Configuracion'
   TextField "Campo de texto_8" at 100,20 size 127x18; Text 'Configuracion de flujo'
   TextField "Campo de texto_9" at 20,48 size 103x15; Text 'Low mass flow cutoff'
   IOField "Campo ES_3" at 159,47 size 96x20
      ProcessValue <- "DB_FLOW_PARA_Setup.Low Massflow cutofff"
   TextField "Campo de texto_10" at 274,47 size 22x15; Text 'kg/s'
   TextField "Campo de texto_1" at 18,79 size 113x15; Text 'Low volume flow cutoff'
   IOField "Campo ES_1" at 158,78 size 96x19; FormatPattern 9.999
      ProcessValue <- "DB_FLOW_PARA_Setup.Low volumeflow cutoff"
   TextField "Campo de texto_2" at 274,81 size 24x15; Text 'm³/s'
   TextField "Campo de texto_3" at 18,105 size 110x15; Text 'Process noise damping'
   SymbolicIOField "Campo ES simbólico_3" at 158,103 size 95x19; TextOn '1'; TextOff '0'; TextList "Process Noise Damping"
      ProcessValue <- "DB_FLOW_PARA_Setup.Process noise damping"
   TextField "Campo de texto_4" at 18,131 size 68x15; Text 'Flow direction'
   SymbolicIOField "Campo ES simbólico_1" at 158,131 size 96x19; TextOn '1'; TextOff '0'; TextList "Flow direction"
      ProcessValue <- "DB_FLOW_PARA_Setup.Flow direction"

screen "120_Zero_Point_Adjust" 320x240, template "Plantilla_1"
   Bar "Barra_1" at 6,150 size 300x30; MinimumValue 0; MaximumValue 100
      ProcessValue <- "DB_FLOW_PARA_Zero Point adjustment.Zero point adjust progress"
   Button "Botón_1" at 54,203 size 52x36; TextOff 'Setup'
      on Click: ActivateScreen("100_Setup", 0)
   Button "Botón_2" at 160,202 size 52x37; TextOff 'Read'
      on Press: SetBit("DB_FLOW_PARA_HMI_Commands.CMD_240")
      on Release: ResetBit("DB_FLOW_PARA_HMI_Commands.CMD_240")
   Button "Botón_3" at 214,202 size 51x37; TextOff 'Start adjustment'
      on Press: SetBit("DB_FLOW_PARA_HMI_Commands.CMD_440")
      on Release: ResetBit("DB_FLOW_PARA_HMI_Commands.CMD_440")
   TextField "Campo de texto_7" at 124,4 size 87x16; Text 'Configuracion'
   TextField "Campo de texto_8" at 100,20 size 121x18; Text 'Ajuste de punto cero'
   TextField "Campo de texto_9" at 15,61 size 80x15; Text 'Zero adjust time'
   IOField "Campo ES_4" at 154,58 size 96x19; FormatPattern 999
      ProcessValue <- "DB_FLOW_PARA_Zero Point adjustment.Zero point duration"
   TextField "Campo de texto_10" at 258,61 size 10x15; Text 's'
   TextField "Campo de texto_1" at 14,93 size 85x15; Text 'Zero offset value'
   IOField "Campo ES_1" at 154,91 size 96x18; FormatPattern s9.99999999
      ProcessValue <- "DB_FLOW_PARA_Zero Point adjustment.Zero point offset value"
   TextField "Campo de texto_2" at 256,92 size 22x15; Text 'kg/s'
   TextField "Campo de texto_3" at 15,121 size 117x15; Text 'Zero standard deviation'
   IOField "Campo ES_2" at 154,121 size 96x17; FormatPattern s9.999999999
      ProcessValue <- "DB_FLOW_PARA_Zero Point adjustment.Standard deviation"
   TextField "Campo de texto_4" at 256,121 size 22x15; Text 'kg/s'

screen "140_Totalizer" 320x240, template "Plantilla_1"
   Button "Botón_1" at 54,202 size 51x37; TextOff 'Setup'
      on Click: ActivateScreen("100_Setup", 0)
   Button "Botón_2" at 159,202 size 53x37; TextOff 'Read'
      on Press: SetBit("DB_FLOW_PARA_HMI_Commands.CMD_220")
      on Release: ResetBit("DB_FLOW_PARA_HMI_Commands.CMD_220")
   Button "Botón_3" at 212,202 size 53x37; TextOff 'Reset totalizer'
      on Press: SetBit("DB_FLOW_PARA_HMI_Commands.CMD_420")
      on Release: ResetBit("DB_FLOW_PARA_HMI_Commands.CMD_420")
   TextField "Campo de texto_7" at 124,4 size 87x16; Text 'Configuracion'
   TextField "Campo de texto_8" at 132,20 size 66x18; Text 'Totalizador'
   TextField "Campo de texto_3" at 44,63 size 48x16; Text 'Totalizer'
   IOField "Campo ES_2" at 146,63 size 96x23; FormatPattern s999999.999
      ProcessValue <- "DB_FLOW_PARA_Totalizer.Totalizer value"
   TextField "Campo de texto_4" at 252,66 size 14x15; Text 'Kg'

screen "200_Identification" 320x240, template "Plantilla_1"
   Button "Botón_1" at 214,202 size 51x37; TextOff 'Read'
      on Press: SetBit("DB_FLOW_PARA_HMI_Commands.CMD_210")
      on Release: ResetBit("DB_FLOW_PARA_HMI_Commands.CMD_210")
   TextField "Campo de texto_7" at 124,4 size 85x16; Text 'Identificacion'
   TextField "Campo de texto_2" at 23,47 size 104x15; Text 'Sensor Serial Number'
   IOField "Campo ES_2" at 164,47 size 121x23; FormatPattern ????????????????????????
      ProcessValue <- "DB_FLOW_PARA_Identification data.Sensor serial number"

screen "300_Operating" 320x240, template "Plantilla_1"
   Button "Botón_1" at 84,60 size 144x35; TextOff 'Varibales de proceso'
      on Click: ActivateScreen("310_Process_Variables", 0)
   TextField "Campo de texto_7" at 128,4 size 63x16; Text 'Operación'
   TextField "Campo de texto_8" at 111,20 size 96x18; Text 'Selección rápida'
   Button "Botón_2" at 84,102 size 144x35; TextOff 'Variables contador'
      on Click: ActivateScreen("320_Contador_Variables", 0)
   Button "Botón_3" at 85,147 size 144x35; TextOff 'Variables principales'
      on Click: ActivateScreen("330_Variables_principales", 0)

screen "310_Process_Variables" 320x240, template "Plantilla_1"
   TextField "Campo de texto_11" at 227,201 size 14x13; Text '°C'
   Button "Botón_1" at 54,203 size 53x36; TextOff 'Operating'
      on Click: ActivateScreen("300_Operating", 0)
   Button "Botón_2" at 160,203 size 52x36; TextOff 'Continious Read'
      on Click: InvertBit("DB_FLOW_PARA_HMI_Commands.CMD_200")
   Button "Botón_3" at 213,203 size 53x36; TextOff 'Single Read'
      on Press: SetBit("DB_FLOW_PARA_HMI_Commands.CMD_200")
      on Release: ResetBit("DB_FLOW_PARA_HMI_Commands.CMD_200")
   TextField "Campo de texto_5" at 128,4 size 63x16; Text 'Operación'
   TextField "Campo de texto_9" at 100,20 size 122x18; Text 'Variables de proceso'
   TextField "Campo de texto_12" at 12,54 size 27x15; Text 'Masa'
   IOField "Campo ES_6" at 105,51 size 96x23; FormatPattern s9.999e
      ProcessValue <- "DB_FLOW_PARA_Process Values.Massflow"
   Button "Botón_9" at 260,51 size 33x22; TextOff 'Text'; PictureOff "png-transparent-pie-chart-computer-icons-graph-of-a-function-others-purple-text-graph-of-a-function"
      on Click: ActivateScreen("311_Mass_Flow_Trend", 0)
   TextField "Campo de texto_1" at 219,55 size 19x13; Text 'kg/s'
   TextField "Campo de texto_7" at 12,82 size 42x15; Text 'Volumen'
   IOField "Campo ES_1" at 104,78 size 96x23; FormatPattern s9.999e
      ProcessValue <- "DB_FLOW_PARA_Process Values.Volumeflow"
   TextField "Campo de texto_2" at 219,83 size 21x13; Text 'm³/s'
   Button "Botón_4" at 261,78 size 32x22; TextOff 'Text'; PictureOff "png-transparent-pie-chart-computer-icons-graph-of-a-function-others-purple-text-graph-of-a-function"
      on Click: ActivateScreen("312_Volume_Flow_Trend", 0)
   TextField "Campo de texto_8" at 12,116 size 46x15; Text 'Densidad'
   TextField "Campo de texto_14" at 219,117 size 27x13; Text 'kg/m³'
   Button "Botón_5" at 260,116 size 33x21; TextOff 'Text'; PictureOff "png-transparent-pie-chart-computer-icons-graph-of-a-function-others-purple-text-graph-of-a-function"
      on Click: ActivateScreen("313_Density_Trend", 0)
   IOField "Campo ES_2" at 105,113 size 96x24; FormatPattern s9999.999
      ProcessValue <- "DB_FLOW_PARA_Process Values.Density"
   TextField "Campo de texto_3" at 11,147 size 64x15; Text 'Temperatura'
   IOField "Campo ES_3" at 105,146 size 96x23; FormatPattern s999.999
      ProcessValue <- "DB_FLOW_PARA_Process Values.Temperature"
   TextField "Campo de texto_10" at 219,150 size 13x13; Text '°C'
   Button "Botón_6" at 259,147 size 34x20; TextOff 'Text'; PictureOff "png-transparent-pie-chart-computer-icons-graph-of-a-function-others-purple-text-graph-of-a-function"
      on Click: ActivateScreen("314_Temperature_Trend", 0)
   TextField "Campo de texto_4" at 3,180 size 93x13; Text 'Marco de temperatura'
   IOField "Campo ES_4" at 105,177 size 96x21; FormatPattern s999.999
      ProcessValue <- "DB_FLOW_PARA_Process Values.Frame temperature"
   Button "Botón_7" at 260,175 size 35x20; TextOff 'Text'; PictureOff "png-transparent-pie-chart-computer-icons-graph-of-a-function-others-purple-text-graph-of-a-function"
      on Click: ActivateScreen("315_Frame_Temperature_Trend", 0)
   TextField "Campo de texto_6" at 219,181 size 13x13; Text '°C'

screen "311_Mass_Flow_Trend" 320x240, template "Plantilla_1"
   TextField "Campo de texto_1" at 8,46 size 68x15; Text 'Current Value'
   IOField "Campo ES_1" at 8,64 size 88x23; FormatPattern s9.999e
      ProcessValue <- "DB_FLOW_PARA_Process Values.Massflow"
   TrendView "Visor de curvas_1" at 109,46 size 206x152
   Button "Botón_1" at 55,202 size 52x37; TextOff 'Operating'
      on Click: ActivateScreen("300_Operating", 0)
   Button "Botón_2" at 108,202 size 52x37; TextOff 'Process Variables'
      on Click: ActivateScreen("310_Process_Variables", 0)
   Button "Botón_3" at 160,202 size 53x37; TextOff 'Continious Read'
      on Click: InvertBit("DB_FLOW_PARA_HMI_Commands.CMD_200")
   Button "Botón_4" at 214,203 size 51x36; TextOff 'Single Read'
      on Press: SetBit("DB_FLOW_PARA_HMI_Commands.CMD_200")
      on Release: ResetBit("DB_FLOW_PARA_HMI_Commands.CMD_200")
   TextField "Campo de texto_5" at 128,0 size 63x16; Text 'Operación'
   TextField "Campo de texto_9" at 80,16 size 165x18; Text 'Variables de proceso - Masa'

screen "312_Volume_Flow_Trend" 320x240, template "Plantilla_1"
   TextField "Campo de texto_2" at 8,47 size 68x15; Text 'Current Value'
   IOField "Campo ES_1" at 3,66 size 95x23; FormatPattern s999999999.999
      ProcessValue <- "DB_FLOW_PARA_Process Values.Volumeflow"
   TrendView "Visor de curvas_1" at 103,48 size 211x150
   Button "Botón_1" at 55,203 size 52x36; TextOff 'Operating'
      on Click: ActivateScreen("300_Operating", 0)
   Button "Botón_2" at 108,203 size 52x36; TextOff 'Process Variables'
      on Click: ActivateScreen("310_Process_Variables", 0)
   Button "Botón_3" at 161,203 size 51x36; TextOff 'Continious Read'
      on Click: InvertBit("DB_FLOW_PARA_HMI_Commands.CMD_200")
   Button "Botón_4" at 214,203 size 51x36; TextOff 'Single Read'
      on Release: ResetBit("DB_FLOW_PARA_HMI_Commands.CMD_200")
      on Press: SetBit("DB_FLOW_PARA_HMI_Commands.CMD_200")
   TextField "Campo de texto_5" at 128,0 size 63x16; Text 'Operación'
   TextField "Campo de texto_9" at 65,16 size 185x18; Text 'Variables de proceso - Volumen'

screen "313_Density_Trend" 320x240, template "Plantilla_1"
   TextField "Campo de texto_2" at 7,52 size 68x15; Text 'Current Value'
   IOField "Campo ES_1" at 7,73 size 102x23; FormatPattern s999999999.999
      ProcessValue <- "DB_FLOW_PARA_Process Values.Density"
   Button "Botón_1" at 55,202 size 51x37; TextOff 'Operating'
      on Click: ActivateScreen("300_Operating", 0)
   Button "Botón_2" at 107,202 size 52x37; TextOff 'Process Variables'
      on Click: ActivateScreen("310_Process_Variables", 0)
   TrendView "Visor de curvas_1" at 113,52 size 202x144
   Button "Botón_3" at 160,202 size 52x37; TextOff 'Continious Read'
      on Click: InvertBit("DB_FLOW_PARA_HMI_Commands.CMD_200")
   Button "Botón_4" at 213,202 size 52x37; TextOff 'Single Read'
      on Release: ResetBit("DB_FLOW_PARA_HMI_Commands.CMD_200")
      on Press: SetBit("DB_FLOW_PARA_HMI_Commands.CMD_200")
   TextField "Campo de texto_5" at 128,0 size 63x16; Text 'Operación'
   TextField "Campo de texto_9" at 65,16 size 187x18; Text 'Variables de proceso - Densidad'

screen "314_Temperature_Trend" 320x240, template "Plantilla_1"
   TextField "Campo de texto_2" at 7,47 size 68x15; Text 'Current Value'
   IOField "Campo ES_1" at 7,63 size 96x23; FormatPattern s999999999.999
      ProcessValue <- "DB_FLOW_PARA_Process Values.Temperature"
   Button "Botón_1" at 55,203 size 51x36; TextOff 'Operating'
      on Click: ActivateScreen("300_Operating", 0)
   Button "Botón_2" at 107,203 size 52x36; TextOff 'Process Variables'
      on Click: ActivateScreen("310_Process_Variables", 0)
   TrendView "Visor de curvas_1" at 111,47 size 205x150
   Button "Botón_3" at 160,203 size 52x36; TextOff 'Continious Read'
      on Click: InvertBit("DB_FLOW_PARA_HMI_Commands.CMD_200")
   Button "Botón_4" at 214,203 size 52x36; TextOff 'Single Read'
      on Release: ResetBit("DB_FLOW_PARA_HMI_Commands.CMD_200")
      on Press: SetBit("DB_FLOW_PARA_HMI_Commands.CMD_200")
   TextField "Campo de texto_5" at 128,0 size 63x16; Text 'Operación'
   TextField "Campo de texto_9" at 65,16 size 210x18; Text 'Variables de proceso - Temperatura'

screen "315_Frame_Temperature_Trend" 320x240, template "Plantilla_1"
   TextField "Campo de texto_2" at 8,51 size 68x15; Text 'Current Value'
   IOField "Campo ES_1" at 6,72 size 96x23; FormatPattern s999999999.999
      ProcessValue <- "DB_FLOW_PARA_Process Values.Temperature"
   Button "Botón_1" at 55,203 size 51x36; TextOff 'Operating'
      on Click: ActivateScreen("300_Operating", 0)
   Button "Botón_2" at 107,203 size 52x36; TextOff 'Process Variables'
      on Click: ActivateScreen("310_Process_Variables", 0)
   TrendView "Visor de curvas_1" at 113,49 size 200x148
   Button "Botón_3" at 161,203 size 51x36; TextOff 'Continious Read'
      on Click: InvertBit("DB_FLOW_PARA_HMI_Commands.CMD_200")
   Button "Botón_4" at 214,203 size 51x36; TextOff 'Single Read'
      on Release: ResetBit("DB_FLOW_PARA_HMI_Commands.CMD_200")
      on Press: SetBit("DB_FLOW_PARA_HMI_Commands.CMD_200")
   TextField "Campo de texto_5" at 128,0 size 63x16; Text 'Operación'
   TextField "Campo de texto_9" at 31,17 size 263x18; Text 'Variables de proceso - Marco de temperatura'

screen "400_Diagnose" 320x240, template "Plantilla_1"
   Button "Botón_1" at 70,69 size 197x36; TextOff 'Device diagnostic'
      on Click: ActivateScreen("410_Device_Diagnostic", 0)
   TextField "Campo de texto_5" at 128,0 size 74x16; Text 'Diagnostico'
   TextField "Campo de texto_9" at 112,16 size 96x18; Text 'Seleccion rapida'

screen "410_Device_Diagnostic" 320x240, template "Plantilla_1"
   Button "Botón_1" at 55,203 size 51x36; TextOff 'Diagnose'
      on Click: ActivateScreen("400_Diagnose", 0)
   TextField "Campo de texto_5" at 128,0 size 74x16; Text 'Diagnostico'
   TextField "Campo de texto_9" at 88,15 size 148x18; Text 'Diagnostico de dispositivo'
   Button "Botón_2" at 212,203 size 53x36; TextOff 'Read'
      on Press: SetBit("DB_FLOW_PARA_HMI_Commands.CMD_230")
      on Release: ResetBit("DB_FLOW_PARA_HMI_Commands.CMD_230")
   TextField "Campo de texto_11" at 49,79 size 94x15; Text 'Pick-up amplitude 1'
   TextField "Campo de texto_12" at 49,127 size 87x15; Text 'Sensor frequency'
   TextField "Campo de texto_13" at 49,105 size 94x15; Text 'Pick-up amplitude 2'
   IOField "Campo ES_5" at 153,79 size 96x23; FormatPattern s999999999.999
      ProcessValue <- "DB_FLOW_PARA_Process Values.Temperature"
   IOField "Campo ES_6" at 153,102 size 96x23; FormatPattern s999999999.999
      ProcessValue <- "DB_FLOW_PARA_Process Values.Temperature"
   IOField "Campo ES_7" at 153,125 size 96x23; FormatPattern s999999999.999
      ProcessValue <- "DB_FLOW_PARA_Process Values.Temperature"
   TextField "Campo de texto_14" at 257,81 size 10x15; Text 'V'
   TextField "Campo de texto_15" at 257,104 size 10x15; Text 'V'
   TextField "Campo de texto_16" at 257,125 size 14x15; Text 'Hz'
   TextField "Campo de texto_1" at 49,56 size 69x15; Text 'Driver current'
   IOField "Campo ES_2" at 153,56 size 96x23; FormatPattern s999999999.999
      ProcessValue <- "DB_FLOW_PARA_Process Values.Temperature"
   TextField "Campo de texto_3" at 257,64 size 10x15; Text 'A'

screen "420_Alarms" 320x240, template "Plantilla_1"
   Button "Botón_1" at 55,203 size 51x36; TextOff 'Diagnose'
      on Click: ActivateScreen("400_Diagnose", 0)
   Button "Botón_2" at 212,203 size 53x36; TextOff 'Read'
      on Release: ResetBit("DB_FLOW_PARA_HMI_Commands.CMD_280")
      on Press: SetBit("DB_FLOW_PARA_HMI_Commands.CMD_280")
   TextField "Campo de texto_5" at 128,0 size 74x16; Text 'Diagnostico'
   TextField "Campo de texto_9" at 140,16 size 49x18; Text 'Alarmas'
   TextField "Campo de texto_3" at 22,53 size 69x15; Text 'Alarm group 1'
   IOField "Campo ES_3" at 156,50 size 138x23; FormatPattern 11111111111111111111111111111111
      ProcessValue <- "DB_FLOW_PARA_Alarms.Alarm group 1"
   TextField "Campo de texto_2" at 15,95 size 140x15; Text 'Alarm group 2 & quality code'
   IOField "Campo ES_1" at 156,90 size 138x23; FormatPattern 11111111111111111111111111111111
      ProcessValue <- "DB_FLOW_PARA_Alarms.Alarm group 2"

screen "320_Contador_Variables" 320x240, template "Plantilla_1"
   TextField "Campo de texto_5" at 128,4 size 63x16; Text 'Operación'
   TextField "Campo de texto_9" at 100,20 size 130x18; Text 'Variables del contador'
   TextField "Campo de texto_2" at 23,59 size 77x15; Text 'Salida secadero'
   IOField "Campo ES_2" at 131,59 size 99x20; FormatPattern 99999
      ProcessValue <- "CONTADOR_DB_cSecadero"
   TextField "Campo de texto_1" at 23,95 size 71x15; Text 'Entrada horno'
   IOField "Campo ES_1" at 131,95 size 99x20; FormatPattern 99999
      ProcessValue <- "CONTADOR_DB_cHorno"
   Button "Botón_9" at 254,57 size 33x22; TextOff 'Text'; PictureOff "png-transparent-pie-chart-computer-icons-graph-of-a-function-others-purple-text-graph-of-a-function"
      on Click: ActivateScreen("311_Mass_Flow_Trend", 0)
   Button "Botón_1" at 254,95 size 33x22; TextOff 'Text'; PictureOff "png-transparent-pie-chart-computer-icons-graph-of-a-function-others-purple-text-graph-of-a-function"
      on Click: ActivateScreen("311_Mass_Flow_Trend", 0)
   Button "Botón_2" at 54,203 size 51x35; TextOff 'Operating'
      on Click: ActivateScreen("300_Operating", 0)

screen "321_Secadero_trend" 320x240, template "Plantilla_1"
   TextField "Campo de texto_5" at 128,3 size 63x16; Text 'Operación'
   TextField "Campo de texto_9" at 43,21 size 225x18; Text 'Variables del contador - Entrada Horno'
   TextField "Campo de texto_2" at 11,52 size 58x15; Text 'Valor actual'
   IOField "Campo ES_1" at 11,67 size 88x23; FormatPattern s99999
      ProcessValue <- "CONTADOR_DB_cHorno"
   TrendView "Visor de curvas_1" at 109,46 size 205x152
   Button "Botón_1" at 54,203 size 51x35; TextOff 'Operating'
      on Click: ActivateScreen("300_Operating", 0)

screen "322_Horno_trend" 320x240, template "Plantilla_1"
   TextField "Campo de texto_5" at 128,0 size 63x16; Text 'Operacion'
   TextField "Campo de texto_9" at 43,21 size 234x18; Text 'Variables del contador - Salida secadero'
   TextField "Campo de texto_2" at 11,52 size 58x15; Text 'Valor actual'
   IOField "Campo ES_1" at 11,67 size 88x23; FormatPattern s99999
      ProcessValue <- "CONTADOR_DB_cSecadero"
   TrendView "Visor de curvas_1" at 109,46 size 205x152
   Button "Botón_1" at 54,203 size 51x35; TextOff 'Operating'
      on Click: ActivateScreen("300_Operating", 0)

screen "330_Variables_principales" 320x240, template "Plantilla_1"
   TextField "Campo de texto_7" at 128,4 size 63x16; Text 'Operación'
   TextField "Campo de texto_1" at 74,99 size 164x18; Text 'Aplicacion engobe y esmalte'
   TextField "Campo de texto_2" at 104,21 size 112x18; Text 'Contador de piezas'
   TextField "Campo de texto_3" at 27,49 size 77x15; Text 'Salida secadero'
   IOField "Campo ES_2" at 110,50 size 99x17; FormatPattern 99999
      ProcessValue <- "CONTADOR_DB_cSecadero"
   Button "Botón_9" at 253,50 size 33x22; TextOff 'Text'; PictureOff "png-transparent-pie-chart-computer-icons-graph-of-a-function-others-purple-text-graph-of-a-function"
      on Click: ActivateScreen("311_Mass_Flow_Trend", 0)
   TextField "Campo de texto_4" at 28,73 size 71x15; Text 'Entrada horno'
   IOField "Campo ES_1" at 110,75 size 99x17; FormatPattern 99999
      ProcessValue <- "CONTADOR_DB_cHorno"
   Button "Botón_1" at 254,74 size 33x22; TextOff 'Text'; PictureOff "png-transparent-pie-chart-computer-icons-graph-of-a-function-others-purple-text-graph-of-a-function"
      on Click: ActivateScreen("311_Mass_Flow_Trend", 0)
   TextField "Campo de texto_8" at 28,125 size 46x15; Text 'Densidad'
   IOField "Campo ES_3" at 110,125 size 98x19; FormatPattern s9999.999
      ProcessValue <- "DB_FLOW_PARA_Process Values.Density"
   TextField "Campo de texto_5" at 28,146 size 64x15; Text 'Temperatura'
   IOField "Campo ES_4" at 110,146 size 97x19; FormatPattern s999.999
      ProcessValue <- "DB_FLOW_PARA_Process Values.Temperature"
   TextField "Campo de texto_14" at 220,122 size 27x13; Text 'kg/m³'
   TextField "Campo de texto_10" at 220,147 size 13x13; Text '°C'
   Button "Botón_5" at 254,123 size 33x21; TextOff 'Text'; PictureOff "png-transparent-pie-chart-computer-icons-graph-of-a-function-others-purple-text-graph-of-a-function"
      on Click: ActivateScreen("313_Density_Trend", 0)
   Button "Botón_6" at 254,145 size 34x20; TextOff 'Text'; PictureOff "png-transparent-pie-chart-computer-icons-graph-of-a-function-others-purple-text-graph-of-a-function"
      on Click: ActivateScreen("314_Temperature_Trend", 0)
   Button "Botón_2" at 54,203 size 53x36; TextOff 'Operating'
      on Click: ActivateScreen("300_Operating", 0)
*)